LIN {X 0,Y 221.494,Z 504.483,A -85,B 0,C 180,E1 -25357.99,E2 -25357.99} C_VEL
LIN {X 0,Y 227.921,Z 439.207,A -85,B 0,C 180,E1 -25359.51,E2 -25359.51} C_VEL
LIN {X 0,Y 226.419,Z 435.193,A -85,B 0,C 180,E1 -25360.912,E2 -25360.912} C_VEL
LIN {X 0,Y 223.343,Z 428.758,A -85,B 0,C 180,E1 -25364.018,E2 -25364.018} C_VEL
LIN {X 0,Y 220.682,Z 423.431,A -85,B 0,C 180,E1 -25367.335,E2 -25367.335} C_VEL
LIN {X 0,Y 218.87,Z 419.91,A -85,B 0,C 180,E1 -25370.237,E2 -25370.237} C_VEL
LIN {X 0,Y 217.27,Z 416.47,A -85,B 0,C 180,E1 -25373.966,E2 -25373.966} C_VEL
LIN {X 0,Y 216.23,Z 414.392,A -85,B 0,C 180,E1 -25380,E2 -25380} C_VEL
LIN {X 0,Y 217.433,Z 416.799,A -85,B 0,C 180,E1 -25386.962,E2 -25386.962} C_VEL
LIN {X 0,Y 219.423,Z 421.023,A -85,B 0,C 180,E1 -25391.197,E2 -25391.197} C_VEL
LIN {X 0,Y 221.498,Z 425.12,A -85,B 0,C 180,E1 -25394.235,E2 -25394.235} C_VEL
LIN {X 0,Y 223.862,Z 429.779,A -85,B 0,C 180,E1 -25397,E2 -25397} C_VEL
LIN {X 0,Y 227.551,Z 437.653,A -85,B 0,C 180,E1 -25400.561,E2 -25400.561} C_VEL
LIN {X 0,Y 227.966,Z 438.553,A -85,B 0,C 180,E1 -25400.919,E2 -25400.919} C_VEL
LIN {X 0,Y 221.714,Z 501.532,A -85,B 0,C 180,E1 -25402.388,E2 -25402.388} C_VEL
LIN {X 0,Y 218.854,Z 518.054,A -85,B 0,C 180,E1 -25402.945,E2 -25402.945} C_VEL
LIN {X 0,Y 214.898,Z 534.172,A -85,B 0,C 180,E1 -25403.694,E2 -25403.694} C_VEL
LIN {X 0,Y 209.854,Z 550.115,A -85,B 0,C 180,E1 -25404.713,E2 -25404.713} C_VEL
LIN {X 0,Y 204.116,Z 564.778,A -85,B 0,C 180,E1 -25405.906,E2 -25405.906} C_VEL
LIN {X 0,Y 197.233,Z 579.446,A -85,B 0,C 180,E1 -25407.461,E2 -25407.461} C_VEL
LIN {X 0,Y 189.58,Z 593.437,A -85,B 0,C 180,E1 -25409.405,E2 -25409.405} C_VEL
LIN {X 0,Y 181.509,Z 606.104,A -85,B 0,C 180,E1 -25411.589,E2 -25411.589} C_VEL
LIN {X 0,Y 173.842,Z 617.019,A -85,B 0,C 180,E1 -25414.028,E2 -25414.028} C_VEL
LIN {X 0,Y 166.48,Z 626.388,A -85,B 0,C 180,E1 -25416.67,E2 -25416.67} C_VEL
LIN {X 0,Y 157.191,Z 637.123,A -85,B 0,C 180,E1 -25420.53,E2 -25420.53} C_VEL
LIN {X 0,Y 148.617,Z 646.133,A -85,B 0,C 180,E1 -25424.819,E2 -25424.819} C_VEL
LIN {X 0,Y 141.063,Z 653.654,A -85,B 0,C 180,E1 -25429.633,E2 -25429.633} C_VEL
LIN {X 0,Y 132.944,Z 661.201,A -85,B 0,C 180,E1 -25436.284,E2 -25436.284} C_VEL
LIN {X 0,Y 126.667,Z 666.92,A -85,B 0,C 180,E1 -25443.649,E2 -25443.649} C_VEL
LIN {X 0,Y 122.985,Z 670.259,A -85,B 0,C 180,E1 -25449.948,E2 -25449.948} C_VEL
LIN {X 0,Y 120.736,Z 672.675,A -85,B 0,C 180,E1 -25456.536,E2 -25456.536} C_VEL
LIN {X 0,Y 119.59,Z 674.038,A -85,B 0,C 180,E1 -25463.25,E2 -25463.25} C_VEL
LIN {X 0,Y 119.419,Z 674.556,A -85,B 0,C 180,E1 -25470,E2 -25470} C_VEL
LIN {X 0,Y 119.59,Z 674.067,A -85,B 0,C 180,E1 -25476.75,E2 -25476.75} C_VEL
LIN {X 0,Y 120.729,Z 672.734,A -85,B 0,C 180,E1 -25483.465,E2 -25483.465} C_VEL
LIN {X 0,Y 122.952,Z 670.346,A -85,B 0,C 180,E1 -25490.057,E2 -25490.057} C_VEL
LIN {X 0,Y 126.618,Z 667.042,A -85,B 0,C 180,E1 -25496.362,E2 -25496.362} C_VEL
LIN {X 0,Y 132.912,Z 661.357,A -85,B 0,C 180,E1 -25503.725,E2 -25503.725} C_VEL
LIN {X 0,Y 141.009,Z 653.864,A -85,B 0,C 180,E1 -25510.385,E2 -25510.385} C_VEL
LIN {X 0,Y 149.586,Z 645.371,A -85,B 0,C 180,E1 -25515.765,E2 -25515.765} C_VEL
LIN {X 0,Y 158.221,Z 636.189,A -85,B 0,C 180,E1 -25520.015,E2 -25520.015} C_VEL
LIN {X 0,Y 166.39,Z 626.732,A -85,B 0,C 180,E1 -25523.371,E2 -25523.371} C_VEL
LIN {X 0,Y 173.745,Z 617.398,A -85,B 0,C 180,E1 -25526.018,E2 -25526.018} C_VEL
LIN {X 0,Y 181.444,Z 606.553,A -85,B 0,C 180,E1 -25528.445,E2 -25528.445} C_VEL
LIN {X 0,Y 189.51,Z 593.974,A -85,B 0,C 180,E1 -25530.632,E2 -25530.632} C_VEL
LIN {X 0,Y 196.444,Z 581.403,A -85,B 0,C 180,E1 -25532.434,E2 -25532.434} C_VEL
LIN {X 0,Y 203.313,Z 567.081,A -85,B 0,C 180,E1 -25533.993,E2 -25533.993} C_VEL
LIN {X 0,Y 209.066,Z 553.002,A -85,B 0,C 180,E1 -25535.179,E2 -25535.179} C_VEL
LIN {X 0,Y 214.072,Z 537.944,A -85,B 0,C 180,E1 -25536.224,E2 -25536.224} C_VEL
LIN {X 0,Y 218.277,Z 521.791,A -85,B 0,C 180,E1 -25537.037,E2 -25537.037} C_VEL
LIN {X 0,Y 221.319,Z 505.505,A -85,B 0,C 180,E1 -25537.631,E2 -25537.631} C_VEL
LIN {X 0,Y 223.9,Z 483.093,A -85,B 0,C 180,E1 -25538.178,E2 -25538.178} C_VEL
LIN {X 0,Y 228.194,Z 438.76,A -85,B 0,C 180,E1 -25539.19,E2 -25539.19} C_VEL
LIN {X 0,Y 224.904,Z 431.726,A -85,B 0,C 180,E1 -25542.261,E2 -25542.261} C_VEL
LIN {X 0,Y 222.442,Z 426.637,A -85,B 0,C 180,E1 -25545.008,E2 -25545.008} C_VEL
LIN {X 0,Y 220.387,Z 422.756,A -85,B 0,C 180,E1 -25547.766,E2 -25547.766} C_VEL
LIN {X 0,Y 219.16,Z 420.172,A -85,B 0,C 180,E1 -25549.841,E2 -25549.841} C_VEL
LIN {X 0,Y 217.586,Z 416.739,A -85,B 0,C 180,E1 -25553.509,E2 -25553.509} C_VEL
LIN {X 0,Y 216.511,Z 414.774,A -85,B 0,C 180,E1 -25560,E2 -25560} C_VEL
LIN {X 0,Y 217.626,Z 416.867,A -85,B 0,C 180,E1 -25566.257,E2 -25566.257} C_VEL
LIN {X 0,Y 219.235,Z 420.273,A -85,B 0,C 180,E1 -25569.922,E2 -25569.922} C_VEL
LIN {X 0,Y 221.587,Z 425.06,A -85,B 0,C 180,E1 -25573.556,E2 -25573.556} C_VEL
LIN {X 0,Y 224.194,Z 430.159,A -85,B 0,C 180,E1 -25576.621,E2 -25576.621} C_VEL
LIN {X 0,Y 227.397,Z 437.132,A -85,B 0,C 180,E1 -25579.757,E2 -25579.757} C_VEL
LIN {X 0,Y 228.202,Z 439.552,A -85,B 0,C 180,E1 -25580.519,E2 -25580.519} C_VEL
LIN {X 0,Y 221.379,Z 507.429,A -85,B 0,C 180,E1 -25582.062,E2 -25582.062} C_VEL
LIN {X 0,Y 218.386,Z 523.964,A -85,B 0,C 180,E1 -25582.589,E2 -25582.589} C_VEL
LIN {X 0,Y 214.635,Z 538.749,A -85,B 0,C 180,E1 -25583.219,E2 -25583.219} C_VEL
LIN {X 0,Y 209.754,Z 553.938,A -85,B 0,C 180,E1 -25584.073,E2 -25584.073} C_VEL
LIN {X 0,Y 203.894,Z 568.874,A -85,B 0,C 180,E1 -25585.204,E2 -25585.204} C_VEL
LIN {X 0,Y 196.702,Z 584.097,A -85,B 0,C 180,E1 -25586.719,E2 -25586.719} C_VEL
LIN {X 0,Y 188.97,Z 598.053,A -85,B 0,C 180,E1 -25588.523,E2 -25588.523} C_VEL
LIN {X 0,Y 181.019,Z 610.686,A -85,B 0,C 180,E1 -25590.642,E2 -25590.642} C_VEL
LIN {X 0,Y 172.227,Z 622.919,A -85,B 0,C 180,E1 -25593.225,E2 -25593.225} C_VEL
LIN {X 0,Y 170.959,Z 624.557,A -85,B 0,C 180,E1 -25593.648,E2 -25593.648} C_VEL
LIN {X 0,Y 167.411,Z 628.624,A -85,B 0,C 180,E1 -25594.531,E2 -25594.531} C_VEL
LIN {X 0,Y 154.654,Z 639.69,A -85,B 0,C 180,E1 -25596.604,E2 -25596.604} C_VEL
LIN {X 0,Y 150.879,Z 643.086,A -85,B 0,C 180,E1 -25597.69,E2 -25597.69} C_VEL
LIN {X 0,Y 149.826,Z 644.194,A -85,B 0,C 180,E1 -25598.15,E2 -25598.15} C_VEL
LIN {X 0,Y 140.813,Z 653.17,A -85,B 0,C 180,E1 -25602.594,E2 -25602.594} C_VEL
LIN {X 0,Y 132.233,Z 661.232,A -85,B 0,C 180,E1 -25608.079,E2 -25608.079} C_VEL
LIN {X 0,Y 125.287,Z 667.51,A -85,B 0,C 180,E1 -25613.915,E2 -25613.915} C_VEL
LIN {X 0,Y 118.796,Z 673.385,A -85,B 0,C 180,E1 -25621.753,E2 -25621.753} C_VEL
LIN {X 0,Y 115.131,Z 676.828,A -85,B 0,C 180,E1 -25628.515,E2 -25628.515} C_VEL
LIN {X 0,Y 112.881,Z 679.342,A -85,B 0,C 180,E1 -25635.58,E2 -25635.58} C_VEL
LIN {X 0,Y 112.089,Z 680.775,A -85,B 0,C 180,E1 -25642.796,E2 -25642.796} C_VEL
LIN {X 0,Y 112.247,Z 681.32,A -85,B 0,C 180,E1 -25650,E2 -25650} C_VEL
LIN {X 0,Y 112.089,Z 680.758,A -85,B 0,C 180,E1 -25657.204,E2 -25657.204} C_VEL
LIN {X 0,Y 112.88,Z 679.308,A -85,B 0,C 180,E1 -25664.421,E2 -25664.421} C_VEL
LIN {X 0,Y 115.126,Z 676.778,A -85,B 0,C 180,E1 -25671.486,E2 -25671.486} C_VEL
LIN {X 0,Y 118.797,Z 673.315,A -85,B 0,C 180,E1 -25678.247,E2 -25678.247} C_VEL
LIN {X 0,Y 125.305,Z 667.419,A -85,B 0,C 180,E1 -25686.08,E2 -25686.08} C_VEL
LIN {X 0,Y 133.826,Z 659.689,A -85,B 0,C 180,E1 -25693.055,E2 -25693.055} C_VEL
LIN {X 0,Y 142.972,Z 650.99,A -85,B 0,C 180,E1 -25698.558,E2 -25698.558} C_VEL
LIN {X 0,Y 152.135,Z 641.463,A -85,B 0,C 180,E1 -25702.957,E2 -25702.957} C_VEL
LIN {X 0,Y 160.614,Z 631.959,A -85,B 0,C 180,E1 -25706.241,E2 -25706.241} C_VEL
LIN {X 0,Y 169.713,Z 620.726,A -85,B 0,C 180,E1 -25709.235,E2 -25709.235} C_VEL
LIN {X 0,Y 177.632,Z 609.886,A -85,B 0,C 180,E1 -25711.438,E2 -25711.438} C_VEL
LIN {X 0,Y 185.662,Z 597.499,A -85,B 0,C 180,E1 -25713.417,E2 -25713.417} C_VEL
LIN {X 0,Y 193.591,Z 583.464,A -85,B 0,C 180,E1 -25715.173,E2 -25715.173} C_VEL
LIN {X 0,Y 200.242,Z 569.835,A -85,B 0,C 180,E1 -25716.479,E2 -25716.479} C_VEL
LIN {X 0,Y 206.156,Z 555.242,A -85,B 0,C 180,E1 -25717.584,E2 -25717.584} C_VEL
LIN {X 0,Y 211.488,Z 539.146,A -85,B 0,C 180,E1 -25718.508,E2 -25718.508} C_VEL
LIN {X 0,Y 215.729,Z 522.746,A -85,B 0,C 180,E1 -25719.158,E2 -25719.158} C_VEL
LIN {X 0,Y 218.588,Z 507.04,A -85,B 0,C 180,E1 -25719.643,E2 -25719.643} C_VEL
LIN {X 0,Y 225.169,Z 442.849,A -85,B 0,C 180,E1 -25721.097,E2 -25721.097} C_VEL
LIN {X 0,Y 222.528,Z 436.715,A -85,B 0,C 180,E1 -25723.84,E2 -25723.84} C_VEL
LIN {X 0,Y 220.247,Z 431.987,A -85,B 0,C 180,E1 -25726.624,E2 -25726.624} C_VEL
LIN {X 0,Y 217.995,Z 427.146,A -85,B 0,C 180,E1 -25730.197,E2 -25730.197} C_VEL
LIN {X 0,Y 216.24,Z 423.391,A -85,B 0,C 180,E1 -25734.405,E2 -25734.405} C_VEL
LIN {X 0,Y 215.36,Z 421.481,A -85,B 0,C 180,E1 -25740,E2 -25740} C_VEL
LIN {X 0,Y 216.439,Z 423.719,A -85,B 0,C 180,E1 -25746.643,E2 -25746.643} C_VEL
LIN {X 0,Y 218.209,Z 427.737,A -85,B 0,C 180,E1 -25750.677,E2 -25750.677} C_VEL
LIN {X 0,Y 220.094,Z 431.665,A -85,B 0,C 180,E1 -25753.621,E2 -25753.621} C_VEL
LIN {X 0,Y 222.294,Z 436.235,A -85,B 0,C 180,E1 -25756.355,E2 -25756.355} C_VEL
LIN {X 0,Y 225.122,Z 442.608,A -85,B 0,C 180,E1 -25759.3,E2 -25759.3} C_VEL
LIN {X 0,Y 219.149,Z 501.479,A -85,B 0,C 180,E1 -25760.669,E2 -25760.669} C_VEL
LIN {X 0,Y 216.266,Z 517.933,A -85,B 0,C 180,E1 -25761.207,E2 -25761.207} C_VEL
LIN {X 0,Y 212.515,Z 533.145,A -85,B 0,C 180,E1 -25761.883,E2 -25761.883} C_VEL
LIN {X 0,Y 207.706,Z 548.35,A -85,B 0,C 180,E1 -25762.775,E2 -25762.775} C_VEL
LIN {X 0,Y 201.845,Z 563.288,A -85,B 0,C 180,E1 -25763.938,E2 -25763.938} C_VEL
LIN {X 0,Y 195.334,Z 577.121,A -85,B 0,C 180,E1 -25765.314,E2 -25765.314} C_VEL
LIN {X 0,Y 187.563,Z 591.314,A -85,B 0,C 180,E1 -25767.138,E2 -25767.138} C_VEL
LIN {X 0,Y 179.949,Z 603.401,A -85,B 0,C 180,E1 -25769.09,E2 -25769.09} C_VEL
LIN {X 0,Y 171.251,Z 615.5,A -85,B 0,C 180,E1 -25771.619,E2 -25771.619} C_VEL
LIN {X 0,Y 163.137,Z 625.599,A -85,B 0,C 180,E1 -25774.327,E2 -25774.327} C_VEL
LIN {X 0,Y 153.81,Z 636.113,A -85,B 0,C 180,E1 -25777.983,E2 -25777.983} C_VEL
LIN {X 0,Y 144.743,Z 645.342,A -85,B 0,C 180,E1 -25782.23,E2 -25782.23} C_VEL
LIN {X 0,Y 135.692,Z 653.865,A -85,B 0,C 180,E1 -25787.676,E2 -25787.676} C_VEL
LIN {X 0,Y 127.055,Z 661.411,A -85,B 0,C 180,E1 -25794.493,E2 -25794.493} C_VEL
LIN {X 0,Y 120.293,Z 667.13,A -85,B 0,C 180,E1 -25802.135,E2 -25802.135} C_VEL
LIN {X 0,Y 116.294,Z 670.469,A -85,B 0,C 180,E1 -25808.74,E2 -25808.74} C_VEL
LIN {X 0,Y 113.824,Z 672.884,A -85,B 0,C 180,E1 -25815.701,E2 -25815.701} C_VEL
LIN {X 0,Y 112.549,Z 674.245,A -85,B 0,C 180,E1 -25822.826,E2 -25822.826} C_VEL
LIN {X 0,Y 112.335,Z 674.763,A -85,B 0,C 180,E1 -25830,E2 -25830} C_VEL
LIN {X 0,Y 112.549,Z 674.274,A -85,B 0,C 180,E1 -25837.174,E2 -25837.174} C_VEL
LIN {X 0,Y 113.801,Z 672.941,A -85,B 0,C 180,E1 -25844.301,E2 -25844.301} C_VEL
LIN {X 0,Y 116.261,Z 670.555,A -85,B 0,C 180,E1 -25851.266,E2 -25851.266} C_VEL
LIN {X 0,Y 120.246,Z 667.25,A -85,B 0,C 180,E1 -25857.877,E2 -25857.877} C_VEL
LIN {X 0,Y 127.025,Z 661.565,A -85,B 0,C 180,E1 -25865.516,E2 -25865.516} C_VEL
LIN {X 0,Y 135.623,Z 654.072,A -85,B 0,C 180,E1 -25872.35,E2 -25872.35} C_VEL
LIN {X 0,Y 144.681,Z 645.578,A -85,B 0,C 180,E1 -25877.797,E2 -25877.797} C_VEL
LIN {X 0,Y 153.719,Z 636.396,A -85,B 0,C 180,E1 -25882.06,E2 -25882.06} C_VEL
LIN {X 0,Y 162.215,Z 626.939,A -85,B 0,C 180,E1 -25885.404,E2 -25885.404} C_VEL
LIN {X 0,Y 169.857,Z 617.604,A -85,B 0,C 180,E1 -25888.016,E2 -25888.016} C_VEL
LIN {X 0,Y 177.814,Z 606.758,A -85,B 0,C 180,E1 -25890.404,E2 -25890.404} C_VEL
LIN {X 0,Y 186.121,Z 594.178,A -85,B 0,C 180,E1 -25892.544,E2 -25892.544} C_VEL
LIN {X 0,Y 193.159,Z 581.779,A -85,B 0,C 180,E1 -25894.283,E2 -25894.283} C_VEL
LIN {X 0,Y 200.304,Z 567.284,A -85,B 0,C 180,E1 -25895.817,E2 -25895.817} C_VEL
LIN {X 0,Y 206.188,Z 553.203,A -85,B 0,C 180,E1 -25896.969,E2 -25896.969} C_VEL
LIN {X 0,Y 211.316,Z 538.142,A -85,B 0,C 180,E1 -25897.982,E2 -25897.982} C_VEL
LIN {X 0,Y 215.622,Z 521.964,A -85,B 0,C 180,E1 -25898.768,E2 -25898.768} C_VEL
LIN {X 0,Y 218.763,Z 505.415,A -85,B 0,C 180,E1 -25899.358,E2 -25899.358} C_VEL
LIN {X 0,Y 221.455,Z 482.343,A -85,B 0,C 180,E1 -25899.904,E2 -25899.904} C_VEL
LIN {X 0,Y 225.371,Z 442.866,A -85,B 0,C 180,E1 -25900.792,E2 -25900.792} C_VEL
LIN {X 0,Y 222.757,Z 436.94,A -85,B 0,C 180,E1 -25903.504,E2 -25903.504} C_VEL
LIN {X 0,Y 220.658,Z 432.526,A -85,B 0,C 180,E1 -25906.062,E2 -25906.062} C_VEL
LIN {X 0,Y 218.91,Z 428.999,A -85,B 0,C 180,E1 -25908.647,E2 -25908.647} C_VEL
LIN {X 0,Y 217.913,Z 426.828,A -85,B 0,C 180,E1 -25910.486,E2 -25910.486} C_VEL
LIN {X 0,Y 216.559,Z 423.625,A -85,B 0,C 180,E1 -25913.945,E2 -25913.945} C_VEL
LIN {X 0,Y 215.643,Z 421.841,A -85,B 0,C 180,E1 -25920,E2 -25920} C_VEL
LIN {X 0,Y 216.664,Z 423.955,A -85,B 0,C 180,E1 -25926.051,E2 -25926.051} C_VEL
LIN {X 0,Y 218.401,Z 427.814,A -85,B 0,C 180,E1 -25930.077,E2 -25930.077} C_VEL
LIN {X 0,Y 220.496,Z 432.245,A -85,B 0,C 180,E1 -25933.361,E2 -25933.361} C_VEL
LIN {X 0,Y 222.814,Z 437.08,A -85,B 0,C 180,E1 -25936.197,E2 -25936.197} C_VEL
LIN {X 0,Y 225.415,Z 443.085,A -85,B 0,C 180,E1 -25938.895,E2 -25938.895} C_VEL
LIN {X 0,Y 218.88,Z 506.754,A -85,B 0,C 180,E1 -25940.325,E2 -25940.325} C_VEL
LIN {X 0,Y 215.741,Z 523.856,A -85,B 0,C 180,E1 -25940.852,E2 -25940.852} C_VEL
LIN {X 0,Y 211.534,Z 539.938,A -85,B 0,C 180,E1 -25941.525,E2 -25941.525} C_VEL
LIN {X 0,Y 206.201,Z 555.726,A -85,B 0,C 180,E1 -25942.407,E2 -25942.407} C_VEL
LIN {X 0,Y 200.222,Z 570.315,A -85,B 0,C 180,E1 -25943.508,E2 -25943.508} C_VEL
LIN {X 0,Y 192.869,Z 585.319,A -85,B 0,C 180,E1 -25944.985,E2 -25944.985} C_VEL
LIN {X 0,Y 184.949,Z 599.026,A -85,B 0,C 180,E1 -25946.75,E2 -25946.75} C_VEL
LIN {X 0,Y 176.591,Z 611.738,A -85,B 0,C 180,E1 -25948.89,E2 -25948.89} C_VEL
LIN {X 0,Y 167.08,Z 624.349,A -85,B 0,C 180,E1 -25951.594,E2 -25951.594} C_VEL
LIN {X 0,Y 158.129,Z 635.109,A -85,B 0,C 180,E1 -25954.693,E2 -25954.693} C_VEL
LIN {X 0,Y 149.826,Z 644.194,A -85,B 0,C 180,E1 -25958.15,E2 -25958.15} C_VEL
LIN {X 0,Y 146.323,Z 647.5,A -85,B 0,C 180,E1 -25959.465,E2 -25959.465} C_VEL
LIN {X 0,Y 139.117,Z 652.656,A -85,B 0,C 180,E1 -25961.254,E2 -25961.254} C_VEL
LIN {X 0,Y 131.8,Z 657.356,A -85,B 0,C 180,E1 -25963.293,E2 -25963.293} C_VEL
LIN {X 0,Y 128.225,Z 659.95,A -85,B 0,C 180,E1 -25965.027,E2 -25965.027} C_VEL
LIN {X 0,Y 119.533,Z 667.3,A -85,B 0,C 180,E1 -25971.877,E2 -25971.877} C_VEL
LIN {X 0,Y 112.473,Z 673.174,A -85,B 0,C 180,E1 -25980.008,E2 -25980.008} C_VEL
LIN {X 0,Y 108.465,Z 676.619,A -85,B 0,C 180,E1 -25987.122,E2 -25987.122} C_VEL
LIN {X 0,Y 105.943,Z 679.133,A -85,B 0,C 180,E1 -25994.612,E2 -25994.612} C_VEL
LIN {X 0,Y 105.012,Z 680.567,A -85,B 0,C 180,E1 -26002.308,E2 -26002.308} C_VEL
LIN {X 0,Y 105.165,Z 681.114,A -85,B 0,C 180,E1 -26010,E2 -26010} C_VEL
LIN {X 0,Y 105.012,Z 680.55,A -85,B 0,C 180,E1 -26017.692,E2 -26017.692} C_VEL
LIN {X 0,Y 105.941,Z 679.098,A -85,B 0,C 180,E1 -26025.388,E2 -26025.388} C_VEL
LIN {X 0,Y 108.461,Z 676.567,A -85,B 0,C 180,E1 -26032.879,E2 -26032.879} C_VEL
LIN {X 0,Y 112.481,Z 673.104,A -85,B 0,C 180,E1 -26039.99,E2 -26039.99} C_VEL
LIN {X 0,Y 119.552,Z 667.208,A -85,B 0,C 180,E1 -26048.116,E2 -26048.116} C_VEL
LIN {X 0,Y 128.647,Z 659.477,A -85,B 0,C 180,E1 -26055.25,E2 -26055.25} C_VEL
LIN {X 0,Y 138.324,Z 650.778,A -85,B 0,C 180,E1 -26060.789,E2 -26060.789} C_VEL
LIN {X 0,Y 148.282,Z 640.876,A -85,B 0,C 180,E1 -26065.337,E2 -26065.337} C_VEL
LIN {X 0,Y 158.052,Z 630.251,A -85,B 0,C 180,E1 -26068.868,E2 -26068.868} C_VEL
LIN {X 0,Y 166.172,Z 620.515,A -85,B 0,C 180,E1 -26071.352,E2 -26071.352} C_VEL
LIN {X 0,Y 174.87,Z 608.891,A -85,B 0,C 180,E1 -26073.659,E2 -26073.659} C_VEL
LIN {X 0,Y 183.288,Z 596.108,A -85,B 0,C 180,E1 -26075.597,E2 -26075.597} C_VEL
LIN {X 0,Y 191.459,Z 581.821,A -85,B 0,C 180,E1 -26077.26,E2 -26077.26} C_VEL
LIN {X 0,Y 198.281,Z 567.923,A -85,B 0,C 180,E1 -26078.499,E2 -26078.499} C_VEL
LIN {X 0,Y 204.155,Z 553.463,A -85,B 0,C 180,E1 -26079.535,E2 -26079.535} C_VEL
LIN {X 0,Y 209.532,Z 537.119,A -85,B 0,C 180,E1 -26080.403,E2 -26080.403} C_VEL
LIN {X 0,Y 213.707,Z 520.692,A -85,B 0,C 180,E1 -26080.99,E2 -26080.99} C_VEL
LIN {X 0,Y 216.555,Z 504.099,A -85,B 0,C 180,E1 -26081.481,E2 -26081.481} C_VEL
LIN {X 0,Y 222.506,Z 446.86,A -85,B 0,C 180,E1 -26082.757,E2 -26082.757} C_VEL
LIN {X 0,Y 219.934,Z 440.86,A -85,B 0,C 180,E1 -26085.78,E2 -26085.78} C_VEL
LIN {X 0,Y 217.832,Z 436.273,A -85,B 0,C 180,E1 -26088.838,E2 -26088.838} C_VEL
LIN {X 0,Y 216.601,Z 433.528,A -85,B 0,C 180,E1 -26091.134,E2 -26091.134} C_VEL
LIN {X 0,Y 215.375,Z 430.464,A -85,B 0,C 180,E1 -26094.382,E2 -26094.382} C_VEL
LIN {X 0,Y 214.489,Z 428.573,A -85,B 0,C 180,E1 -26100,E2 -26100} C_VEL
LIN {X 0,Y 215.414,Z 430.565,A -85,B 0,C 180,E1 -26106.204,E2 -26106.204} C_VEL
LIN {X 0,Y 217.153,Z 434.775,A -85,B 0,C 180,E1 -26110.42,E2 -26110.42} C_VEL
LIN {X 0,Y 218.792,Z 438.383,A -85,B 0,C 180,E1 -26113.113,E2 -26113.113} C_VEL
LIN {X 0,Y 220.845,Z 442.924,A -85,B 0,C 180,E1 -26115.813,E2 -26115.813} C_VEL
LIN {X 0,Y 222.485,Z 446.827,A -85,B 0,C 180,E1 -26117.678,E2 -26117.678} C_VEL
LIN {X 0,Y 216.748,Z 501.746,A -85,B 0,C 180,E1 -26118.92,E2 -26118.92} C_VEL
LIN {X 0,Y 213.865,Z 517.845,A -85,B 0,C 180,E1 -26119.423,E2 -26119.423} C_VEL
LIN {X 0,Y 209.968,Z 533.394,A -85,B 0,C 180,E1 -26120.09,E2 -26120.09} C_VEL
LIN {X 0,Y 205.061,Z 548.564,A -85,B 0,C 180,E1 -26120.945,E2 -26120.945} C_VEL
LIN {X 0,Y 199.072,Z 563.501,A -85,B 0,C 180,E1 -26122.071,E2 -26122.071} C_VEL
LIN {X 0,Y 192.397,Z 577.334,A -85,B 0,C 180,E1 -26123.397,E2 -26123.397} C_VEL
LIN {X 0,Y 184.422,Z 591.526,A -85,B 0,C 180,E1 -26125.168,E2 -26125.168} C_VEL
LIN {X 0,Y 176.597,Z 603.612,A -85,B 0,C 180,E1 -26127.071,E2 -26127.071} C_VEL
LIN {X 0,Y 167.628,Z 615.711,A -85,B 0,C 180,E1 -26129.546,E2 -26129.546} C_VEL
LIN {X 0,Y 159.61,Z 625.33,A -85,B 0,C 180,E1 -26132.04,E2 -26132.04} C_VEL
LIN {X 0,Y 150.74,Z 635.095,A -85,B 0,C 180,E1 -26135.323,E2 -26135.323} C_VEL
LIN {X 0,Y 141.169,Z 644.459,A -85,B 0,C 180,E1 -26139.497,E2 -26139.497} C_VEL
LIN {X 0,Y 132.484,Z 652.288,A -85,B 0,C 180,E1 -26144.263,E2 -26144.263} C_VEL
LIN {X 0,Y 124.735,Z 658.814,A -85,B 0,C 180,E1 -26149.613,E2 -26149.613} C_VEL
LIN {X 0,Y 118.132,Z 664.087,A -85,B 0,C 180,E1 -26155.585,E2 -26155.585} C_VEL
LIN {X 0,Y 114.014,Z 667.34,A -85,B 0,C 180,E1 -26160.454,E2 -26160.454} C_VEL
LIN {X 0,Y 109.667,Z 670.678,A -85,B 0,C 180,E1 -26167.387,E2 -26167.387} C_VEL
LIN {X 0,Y 106.915,Z 673.093,A -85,B 0,C 180,E1 -26174.755,E2 -26174.755} C_VEL
LIN {X 0,Y 105.5,Z 674.453,A -85,B 0,C 180,E1 -26182.343,E2 -26182.343} C_VEL
LIN {X 0,Y 105.237,Z 674.97,A -85,B 0,C 180,E1 -26190,E2 -26190} C_VEL
LIN {X 0,Y 105.499,Z 674.481,A -85,B 0,C 180,E1 -26197.656,E2 -26197.656} C_VEL
LIN {X 0,Y 106.895,Z 673.15,A -85,B 0,C 180,E1 -26205.247,E2 -26205.247} C_VEL
LIN {X 0,Y 109.635,Z 670.763,A -85,B 0,C 180,E1 -26212.62,E2 -26212.62} C_VEL
LIN {X 0,Y 113.969,Z 667.458,A -85,B 0,C 180,E1 -26219.559,E2 -26219.559} C_VEL
LIN {X 0,Y 121.259,Z 661.773,A -85,B 0,C 180,E1 -26227.485,E2 -26227.485} C_VEL
LIN {X 0,Y 130.404,Z 654.28,A -85,B 0,C 180,E1 -26234.476,E2 -26234.476} C_VEL
LIN {X 0,Y 139.97,Z 645.786,A -85,B 0,C 180,E1 -26239.97,E2 -26239.97} C_VEL
LIN {X 0,Y 149.419,Z 636.603,A -85,B 0,C 180,E1 -26244.228,E2 -26244.228} C_VEL
LIN {X 0,Y 158.247,Z 627.146,A -85,B 0,C 180,E1 -26247.545,E2 -26247.545} C_VEL
LIN {X 0,Y 167.542,Z 616.114,A -85,B 0,C 180,E1 -26250.506,E2 -26250.506} C_VEL
LIN {X 0,Y 175.83,Z 605.021,A -85,B 0,C 180,E1 -26252.789,E2 -26252.789} C_VEL
LIN {X 0,Y 183.633,Z 593.216,A -85,B 0,C 180,E1 -26254.711,E2 -26254.711} C_VEL
LIN {X 0,Y 190.831,Z 580.83,A -85,B 0,C 180,E1 -26256.349,E2 -26256.349} C_VEL
LIN {X 0,Y 198.248,Z 565.909,A -85,B 0,C 180,E1 -26257.84,E2 -26257.84} C_VEL
LIN {X 0,Y 204.259,Z 551.424,A -85,B 0,C 180,E1 -26258.953,E2 -26258.953} C_VEL
LIN {X 0,Y 209.527,Z 535.745,A -85,B 0,C 180,E1 -26259.913,E2 -26259.913} C_VEL
LIN {X 0,Y 213.648,Z 520.09,A -85,B 0,C 180,E1 -26260.617,E2 -26260.617} C_VEL
LIN {X 0,Y 216.735,Z 503.437,A -85,B 0,C 180,E1 -26261.172,E2 -26261.172} C_VEL
LIN {X 0,Y 221.477,Z 459.215,A -85,B 0,C 180,E1 -26262.169,E2 -26262.169} C_VEL
LIN {X 0,Y 222.725,Z 446.978,A -85,B 0,C 180,E1 -26262.437,E2 -26262.437} C_VEL
LIN {X 0,Y 219.947,Z 440.496,A -85,B 0,C 180,E1 -26265.751,E2 -26265.751} C_VEL
LIN {X 0,Y 218.02,Z 436.399,A -85,B 0,C 180,E1 -26268.6,E2 -26268.6} C_VEL
LIN {X 0,Y 216.807,Z 433.658,A -85,B 0,C 180,E1 -26270.907,E2 -26270.907} C_VEL
LIN {X 0,Y 215.541,Z 430.546,A -85,B 0,C 180,E1 -26274.386,E2 -26274.386} C_VEL
LIN {X 0,Y 214.776,Z 428.903,A -85,B 0,C 180,E1 -26280,E2 -26280} C_VEL
LIN {X 0,Y 215.676,Z 430.896,A -85,B 0,C 180,E1 -26285.727,E2 -26285.727} C_VEL
LIN {X 0,Y 217.325,Z 434.793,A -85,B 0,C 180,E1 -26289.775,E2 -26289.775} C_VEL
LIN {X 0,Y 219.513,Z 439.612,A -85,B 0,C 180,E1 -26293.304,E2 -26293.304} C_VEL
LIN {X 0,Y 221.933,Z 445.082,A -85,B 0,C 180,E1 -26296.322,E2 -26296.322} C_VEL
LIN {X 0,Y 222.764,Z 447.124,A -85,B 0,C 180,E1 -26297.245,E2 -26297.245} C_VEL
LIN {X 0,Y 216.525,Z 506.54,A -85,B 0,C 180,E1 -26298.567,E2 -26298.567} C_VEL
LIN {X 0,Y 213.335,Z 523.559,A -85,B 0,C 180,E1 -26299.063,E2 -26299.063} C_VEL
LIN {X 0,Y 209.025,Z 539.738,A -85,B 0,C 180,E1 -26299.707,E2 -26299.707} C_VEL
LIN {X 0,Y 203.561,Z 555.617,A -85,B 0,C 180,E1 -26300.563,E2 -26300.563} C_VEL
LIN {X 0,Y 197.487,Z 570.112,A -85,B 0,C 180,E1 -26301.611,E2 -26301.611} C_VEL
LIN {X 0,Y 189.967,Z 585.116,A -85,B 0,C 180,E1 -26303.036,E2 -26303.036} C_VEL
LIN {X 0,Y 181.845,Z 598.821,A -85,B 0,C 180,E1 -26304.739,E2 -26304.739} C_VEL
LIN {X 0,Y 173.239,Z 611.532,A -85,B 0,C 180,E1 -26306.812,E2 -26306.812} C_VEL
LIN {X 0,Y 163.436,Z 624.142,A -85,B 0,C 180,E1 -26309.451,E2 -26309.451} C_VEL
LIN {X 0,Y 154.144,Z 634.901,A -85,B 0,C 180,E1 -26312.491,E2 -26312.491} C_VEL
LIN {X 0,Y 144.65,Z 644.844,A -85,B 0,C 180,E1 -26316.279,E2 -26316.279} C_VEL
LIN {X 0,Y 134.935,Z 653.979,A -85,B 0,C 180,E1 -26320.956,E2 -26320.956} C_VEL
LIN {X 0,Y 128.225,Z 659.95,A -85,B 0,C 180,E1 -26325.027,E2 -26325.027} C_VEL
LIN {X 0,Y 124.771,Z 662.455,A -85,B 0,C 180,E1 -26326.897,E2 -26326.897} C_VEL
LIN {X 0,Y 112.428,Z 668.953,A -85,B 0,C 180,E1 -26332.287,E2 -26332.287} C_VEL
LIN {X 0,Y 109.113,Z 670.83,A -85,B 0,C 180,E1 -26334.625,E2 -26334.625} C_VEL
LIN {X 0,Y 108.273,Z 671.396,A -85,B 0,C 180,E1 -26335.512,E2 -26335.512} C_VEL
LIN {X 0,Y 103.922,Z 674.808,A -85,B 0,C 180,E1 -26341.746,E2 -26341.746} C_VEL
LIN {X 0,Y 100.267,Z 677.781,A -85,B 0,C 180,E1 -26349.485,E2 -26349.485} C_VEL
LIN {X 0,Y 98.31,Z 679.756,A -85,B 0,C 180,E1 -26357.616,E2 -26357.616} C_VEL
LIN {X 0,Y 97.902,Z 680.744,A -85,B 0,C 180,E1 -26365.884,E2 -26365.884} C_VEL
LIN {X 0,Y 98.07,Z 680.906,A -85,B 0,C 180,E1 -26370,E2 -26370} C_VEL
LIN {X 0,Y 97.931,Z 680.341,A -85,B 0,C 180,E1 -26378.252,E2 -26378.252} C_VEL
LIN {X 0,Y 99.039,Z 678.888,A -85,B 0,C 180,E1 -26386.49,E2 -26386.49} C_VEL
LIN {X 0,Y 101.873,Z 676.357,A -85,B 0,C 180,E1 -26394.452,E2 -26394.452} C_VEL
LIN {X 0,Y 106.302,Z 672.892,A -85,B 0,C 180,E1 -26401.932,E2 -26401.932} C_VEL
LIN {X 0,Y 113.974,Z 666.996,A -85,B 0,C 180,E1 -26410.35,E2 -26410.35} C_VEL
LIN {X 0,Y 123.685,Z 659.265,A -85,B 0,C 180,E1 -26417.619,E2 -26417.619} C_VEL
LIN {X 0,Y 133.905,Z 650.567,A -85,B 0,C 180,E1 -26423.167,E2 -26423.167} C_VEL
LIN {X 0,Y 143.683,Z 641.264,A -85,B 0,C 180,E1 -26427.45,E2 -26427.45} C_VEL
LIN {X 0,Y 153.101,Z 631.535,A -85,B 0,C 180,E1 -26430.713,E2 -26430.713} C_VEL
LIN {X 0,Y 162.871,Z 620.304,A -85,B 0,C 180,E1 -26433.556,E2 -26433.556} C_VEL
LIN {X 0,Y 172.641,Z 607.57,A -85,B 0,C 180,E1 -26435.979,E2 -26435.979} C_VEL
LIN {X 0,Y 181.961,Z 593.54,A -85,B 0,C 180,E1 -26437.966,E2 -26437.966} C_VEL
LIN {X 0,Y 190.348,Z 578.746,A -85,B 0,C 180,E1 -26439.535,E2 -26439.535} C_VEL
LIN {X 0,Y 197.311,Z 564.167,A -85,B 0,C 180,E1 -26440.716,E2 -26440.716} C_VEL
LIN {X 0,Y 203.604,Z 548.173,A -85,B 0,C 180,E1 -26441.714,E2 -26441.714} C_VEL
LIN {X 0,Y 208.506,Z 532.663,A -85,B 0,C 180,E1 -26442.412,E2 -26442.412} C_VEL
LIN {X 0,Y 212.486,Z 515.86,A -85,B 0,C 180,E1 -26442.954,E2 -26442.954} C_VEL
LIN {X 0,Y 215.119,Z 498.264,A -85,B 0,C 180,E1 -26443.404,E2 -26443.404} C_VEL
LIN {X 0,Y 220.043,Z 451.149,A -85,B 0,C 180,E1 -26444.415,E2 -26444.415} C_VEL
LIN {X 0,Y 217.815,Z 445.762,A -85,B 0,C 180,E1 -26447.398,E2 -26447.398} C_VEL
LIN {X 0,Y 215.936,Z 441.365,A -85,B 0,C 180,E1 -26450.635,E2 -26450.635} C_VEL
LIN {X 0,Y 214.357,Z 437.386,A -85,B 0,C 180,E1 -26454.827,E2 -26454.827} C_VEL
LIN {X 0,Y 213.62,Z 435.652,A -85,B 0,C 180,E1 -26460,E2 -26460} C_VEL
LIN {X 0,Y 214.428,Z 437.543,A -85,B 0,C 180,E1 -26465.879,E2 -26465.879} C_VEL
LIN {X 0,Y 215.998,Z 441.585,A -85,B 0,C 180,E1 -26469.96,E2 -26469.96} C_VEL
LIN {X 0,Y 217.584,Z 445.253,A -85,B 0,C 180,E1 -26472.712,E2 -26472.712} C_VEL
LIN {X 0,Y 219.464,Z 449.769,A -85,B 0,C 180,E1 -26475.33,E2 -26475.33} C_VEL
LIN {X 0,Y 220.013,Z 451.106,A -85,B 0,C 180,E1 -26476.009,E2 -26476.009} C_VEL
LIN {X 0,Y 214.448,Z 502.776,A -85,B 0,C 180,E1 -26477.148,E2 -26477.148} C_VEL
LIN {X 0,Y 211.304,Z 519.519,A -85,B 0,C 180,E1 -26477.661,E2 -26477.661} C_VEL
LIN {X 0,Y 207.268,Z 534.818,A -85,B 0,C 180,E1 -26478.303,E2 -26478.303} C_VEL
LIN {X 0,Y 201.879,Z 550.755,A -85,B 0,C 180,E1 -26479.214,E2 -26479.214} C_VEL
LIN {X 0,Y 195.751,Z 565.415,A -85,B 0,C 180,E1 -26480.29,E2 -26480.29} C_VEL
LIN {X 0,Y 188.317,Z 580.148,A -85,B 0,C 180,E1 -26481.703,E2 -26481.703} C_VEL
LIN {X 0,Y 180.045,Z 594.073,A -85,B 0,C 180,E1 -26483.464,E2 -26483.464} C_VEL
LIN {X 0,Y 171.285,Z 606.737,A -85,B 0,C 180,E1 -26485.488,E2 -26485.488} C_VEL
LIN {X 0,Y 162.829,Z 617.652,A -85,B 0,C 180,E1 -26487.772,E2 -26487.772} C_VEL
LIN {X 0,Y 154.604,Z 627.023,A -85,B 0,C 180,E1 -26490.266,E2 -26490.266} C_VEL
LIN {X 0,Y 144.171,Z 637.756,A -85,B 0,C 180,E1 -26494.034,E2 -26494.034} C_VEL
LIN {X 0,Y 134.356,Z 646.765,A -85,B 0,C 180,E1 -26498.314,E2 -26498.314} C_VEL
LIN {X 0,Y 125.453,Z 654.287,A -85,B 0,C 180,E1 -26503.258,E2 -26503.258} C_VEL
LIN {X 0,Y 115.69,Z 661.832,A -85,B 0,C 180,E1 -26510.368,E2 -26510.368} C_VEL
LIN {X 0,Y 107.852,Z 667.549,A -85,B 0,C 180,E1 -26518.58,E2 -26518.58} C_VEL
LIN {X 0,Y 103.116,Z 670.887,A -85,B 0,C 180,E1 -26525.862,E2 -26525.862} C_VEL
LIN {X 0,Y 100.05,Z 673.302,A -85,B 0,C 180,E1 -26533.681,E2 -26533.681} C_VEL
LIN {X 0,Y 98.457,Z 674.661,A -85,B 0,C 180,E1 -26541.792,E2 -26541.792} C_VEL
LIN {X 0,Y 98.15,Z 675.177,A -85,B 0,C 180,E1 -26550,E2 -26550} C_VEL
LIN {X 0,Y 98.456,Z 674.689,A -85,B 0,C 180,E1 -26558.208,E2 -26558.208} C_VEL
LIN {X 0,Y 100.032,Z 673.358,A -85,B 0,C 180,E1 -26566.321,E2 -26566.321} C_VEL
LIN {X 0,Y 103.085,Z 670.97,A -85,B 0,C 180,E1 -26574.146,E2 -26574.146} C_VEL
LIN {X 0,Y 107.807,Z 667.666,A -85,B 0,C 180,E1 -26581.434,E2 -26581.434} C_VEL
LIN {X 0,Y 115.663,Z 661.981,A -85,B 0,C 180,E1 -26589.643,E2 -26589.643} C_VEL
LIN {X 0,Y 125.388,Z 654.488,A -85,B 0,C 180,E1 -26596.773,E2 -26596.773} C_VEL
LIN {X 0,Y 134.295,Z 646.991,A -85,B 0,C 180,E1 -26601.719,E2 -26601.719} C_VEL
LIN {X 0,Y 144.084,Z 638.031,A -85,B 0,C 180,E1 -26606.017,E2 -26606.017} C_VEL
LIN {X 0,Y 154.53,Z 627.353,A -85,B 0,C 180,E1 -26609.781,E2 -26609.781} C_VEL
LIN {X 0,Y 164.147,Z 616.319,A -85,B 0,C 180,E1 -26612.674,E2 -26612.674} C_VEL
LIN {X 0,Y 172.696,Z 605.226,A -85,B 0,C 180,E1 -26614.887,E2 -26614.887} C_VEL
LIN {X 0,Y 180.699,Z 593.421,A -85,B 0,C 180,E1 -26616.758,E2 -26616.758} C_VEL
LIN {X 0,Y 188.041,Z 581.12,A -85,B 0,C 180,E1 -26618.325,E2 -26618.325} C_VEL
LIN {X 0,Y 195.685,Z 566.111,A -85,B 0,C 180,E1 -26619.763,E2 -26619.763} C_VEL
LIN {X 0,Y 201.818,Z 551.625,A -85,B 0,C 180,E1 -26620.835,E2 -26620.835} C_VEL
LIN {X 0,Y 207.197,Z 535.943,A -85,B 0,C 180,E1 -26621.756,E2 -26621.756} C_VEL
LIN {X 0,Y 211.367,Z 520.451,A -85,B 0,C 180,E1 -26622.423,E2 -26622.423} C_VEL
LIN {X 0,Y 214.609,Z 503.331,A -85,B 0,C 180,E1 -26622.967,E2 -26622.967} C_VEL
LIN {X 0,Y 220.268,Z 451.303,A -85,B 0,C 180,E1 -26624.092,E2 -26624.092} C_VEL
LIN {X 0,Y 218.129,Z 446.088,A -85,B 0,C 180,E1 -26626.965,E2 -26626.965} C_VEL
LIN {X 0,Y 215.933,Z 440.871,A -85,B 0,C 180,E1 -26630.87,E2 -26630.87} C_VEL
LIN {X 0,Y 214.535,Z 437.47,A -85,B 0,C 180,E1 -26634.831,E2 -26634.831} C_VEL
LIN {X 0,Y 213.908,Z 435.972,A -85,B 0,C 180,E1 -26640,E2 -26640} C_VEL
LIN {X 0,Y 214.696,Z 437.842,A -85,B 0,C 180,E1 -26645.4,E2 -26645.4} C_VEL
LIN {X 0,Y 216.141,Z 441.517,A -85,B 0,C 180,E1 -26649.238,E2 -26649.238} C_VEL
LIN {X 0,Y 217.826,Z 445.478,A -85,B 0,C 180,E1 -26652.224,E2 -26652.224} C_VEL
LIN {X 0,Y 219.867,Z 450.363,A -85,B 0,C 180,E1 -26655.053,E2 -26655.053} C_VEL
LIN {X 0,Y 220.292,Z 451.358,A -85,B 0,C 180,E1 -26655.57,E2 -26655.57} C_VEL
LIN {X 0,Y 214.305,Z 506.748,A -85,B 0,C 180,E1 -26656.773,E2 -26656.773} C_VEL
LIN {X 0,Y 210.904,Z 524.382,A -85,B 0,C 180,E1 -26657.274,E2 -26657.274} C_VEL
LIN {X 0,Y 206.414,Z 540.607,A -85,B 0,C 180,E1 -26657.901,E2 -26657.901} C_VEL
LIN {X 0,Y 201.127,Z 555.527,A -85,B 0,C 180,E1 -26658.671,E2 -26658.671} C_VEL
LIN {X 0,Y 194.973,Z 569.909,A -85,B 0,C 180,E1 -26659.663,E2 -26659.663} C_VEL
LIN {X 0,Y 187.295,Z 584.912,A -85,B 0,C 180,E1 -26661.03,E2 -26661.03} C_VEL
LIN {X 0,Y 178.974,Z 598.616,A -85,B 0,C 180,E1 -26662.662,E2 -26662.662} C_VEL
LIN {X 0,Y 170.89,Z 610.308,A -85,B 0,C 180,E1 -26664.481,E2 -26664.481} C_VEL
LIN {X 0,Y 161.458,Z 622.299,A -85,B 0,C 180,E1 -26666.833,E2 -26666.833} C_VEL
LIN {X 0,Y 151.769,Z 633.256,A -85,B 0,C 180,E1 -26669.744,E2 -26669.744} C_VEL
LIN {X 0,Y 142.525,Z 642.608,A -85,B 0,C 180,E1 -26673.042,E2 -26673.042} C_VEL
LIN {X 0,Y 133.892,Z 650.719,A -85,B 0,C 180,E1 -26676.826,E2 -26676.826} C_VEL
LIN {X 0,Y 123.667,Z 659.396,A -85,B 0,C 180,E1 -26682.372,E2 -26682.372} C_VEL
LIN {X 0,Y 113.954,Z 667.091,A -85,B 0,C 180,E1 -26689.641,E2 -26689.641} C_VEL
LIN {X 0,Y 108.273,Z 671.396,A -85,B 0,C 180,E1 -26695.512,E2 -26695.512} C_VEL
LIN {X 0,Y 105.508,Z 673.109,A -85,B 0,C 180,E1 -26698.169,E2 -26698.169} C_VEL
LIN {X 0,Y 99.744,Z 675.475,A -85,B 0,C 180,E1 -26702.482,E2 -26702.482} C_VEL
LIN {X 0,Y 95.371,Z 677.04,A -85,B 0,C 180,E1 -26706.286,E2 -26706.286} C_VEL
LIN {X 0,Y 93.066,Z 678.006,A -85,B 0,C 180,E1 -26709.553,E2 -26709.553} C_VEL
LIN {X 0,Y 92.608,Z 678.314,A -85,B 0,C 180,E1 -26710.723,E2 -26710.723} C_VEL
LIN {X 0,Y 90.855,Z 680.15,A -85,B 0,C 180,E1 -26721.1,E2 -26721.1} C_VEL
LIN {X 0,Y 90.968,Z 680.699,A -85,B 0,C 180,E1 -26730,E2 -26730} C_VEL
LIN {X 0,Y 90.855,Z 680.132,A -85,B 0,C 180,E1 -26738.9,E2 -26738.9} C_VEL
LIN {X 0,Y 92.178,Z 678.678,A -85,B 0,C 180,E1 -26747.757,E2 -26747.757} C_VEL
LIN {X 0,Y 95.377,Z 676.146,A -85,B 0,C 180,E1 -26756.239,E2 -26756.239} C_VEL
LIN {X 0,Y 100.253,Z 672.681,A -85,B 0,C 180,E1 -26764.113,E2 -26764.113} C_VEL
LIN {X 0,Y 108.566,Z 666.784,A -85,B 0,C 180,E1 -26772.821,E2 -26772.821} C_VEL
LIN {X 0,Y 118.94,Z 659.053,A -85,B 0,C 180,E1 -26780.188,E2 -26780.188} C_VEL
LIN {X 0,Y 129.72,Z 650.356,A -85,B 0,C 180,E1 -26785.711,E2 -26785.711} C_VEL
LIN {X 0,Y 139.244,Z 641.692,A -85,B 0,C 180,E1 -26789.687,E2 -26789.687} C_VEL
LIN {X 0,Y 149.71,Z 631.323,A -85,B 0,C 180,E1 -26793.117,E2 -26793.117} C_VEL
LIN {X 0,Y 159.82,Z 620.093,A -85,B 0,C 180,E1 -26795.848,E2 -26795.848} C_VEL
LIN {X 0,Y 169.327,Z 608.071,A -85,B 0,C 180,E1 -26798.066,E2 -26798.066} C_VEL
LIN {X 0,Y 178.628,Z 594.505,A -85,B 0,C 180,E1 -26799.941,E2 -26799.941} C_VEL
LIN {X 0,Y 186.404,Z 581.395,A -85,B 0,C 180,E1 -26801.313,E2 -26801.313} C_VEL
LIN {X 0,Y 193.508,Z 567.495,A -85,B 0,C 180,E1 -26802.433,E2 -26802.433} C_VEL
LIN {X 0,Y 199.451,Z 553.474,A -85,B 0,C 180,E1 -26803.337,E2 -26803.337} C_VEL
LIN {X 0,Y 204.639,Z 538.499,A -85,B 0,C 180,E1 -26804.073,E2 -26804.073} C_VEL
LIN {X 0,Y 209.103,Z 522.081,A -85,B 0,C 180,E1 -26804.619,E2 -26804.619} C_VEL
LIN {X 0,Y 212.112,Z 506.37,A -85,B 0,C 180,E1 -26805.054,E2 -26805.054} C_VEL
LIN {X 0,Y 217.744,Z 455.535,A -85,B 0,C 180,E1 -26806.12,E2 -26806.12} C_VEL
LIN {X 0,Y 215.642,Z 450.223,A -85,B 0,C 180,E1 -26809.437,E2 -26809.437} C_VEL
LIN {X 0,Y 214.314,Z 446.984,A -85,B 0,C 180,E1 -26812.226,E2 -26812.226} C_VEL
LIN {X 0,Y 213.354,Z 444.286,A -85,B 0,C 180,E1 -26815.277,E2 -26815.277} C_VEL
LIN {X 0,Y 212.745,Z 442.779,A -85,B 0,C 180,E1 -26820.473,E2 -26820.473} C_VEL
LIN {X 0,Y 213.481,Z 444.602,A -85,B 0,C 180,E1 -26825.668,E2 -26825.668} C_VEL
LIN {X 0,Y 214.864,Z 448.352,A -85,B 0,C 180,E1 -26829.496,E2 -26829.496} C_VEL
LIN {X 0,Y 216.384,Z 452.146,A -85,B 0,C 180,E1 -26832.307,E2 -26832.307} C_VEL
LIN {X 0,Y 217.698,Z 455.45,A -85,B 0,C 180,E1 -26834.276,E2 -26834.276} C_VEL
LIN {X 0,Y 212.693,Z 501.27,A -85,B 0,C 180,E1 -26835.281,E2 -26835.281} C_VEL
LIN {X 0,Y 209.638,Z 517.993,A -85,B 0,C 180,E1 -26835.754,E2 -26835.754} C_VEL
LIN {X 0,Y 205.511,Z 533.901,A -85,B 0,C 180,E1 -26836.384,E2 -26836.384} C_VEL
LIN {X 0,Y 200.427,Z 548.991,A -85,B 0,C 180,E1 -26837.153,E2 -26837.153} C_VEL
LIN {X 0,Y 194.19,Z 563.926,A -85,B 0,C 180,E1 -26838.192,E2 -26838.192} C_VEL
LIN {X 0,Y 187.206,Z 577.758,A -85,B 0,C 180,E1 -26839.4,E2 -26839.4} C_VEL
LIN {X 0,Y 178.822,Z 591.95,A -85,B 0,C 180,E1 -26841.028,E2 -26841.028} C_VEL
LIN {X 0,Y 169.849,Z 605.006,A -85,B 0,C 180,E1 -26842.978,E2 -26842.978} C_VEL
LIN {X 0,Y 161.074,Z 616.133,A -85,B 0,C 180,E1 -26845.128,E2 -26845.128} C_VEL
LIN {X 0,Y 151.116,Z 627.235,A -85,B 0,C 180,E1 -26847.916,E2 -26847.916} C_VEL
LIN {X 0,Y 140.298,Z 637.966,A -85,B 0,C 180,E1 -26851.616,E2 -26851.616} C_VEL
LIN {X 0,Y 130.034,Z 646.976,A -85,B 0,C 180,E1 -26855.835,E2 -26855.835} C_VEL
LIN {X 0,Y 120.65,Z 654.498,A -85,B 0,C 180,E1 -26860.777,E2 -26860.777} C_VEL
LIN {X 0,Y 110.262,Z 662.042,A -85,B 0,C 180,E1 -26867.99,E2 -26867.99} C_VEL
LIN {X 0,Y 101.819,Z 667.759,A -85,B 0,C 180,E1 -26876.482,E2 -26876.482} C_VEL
LIN {X 0,Y 96.65,Z 671.096,A -85,B 0,C 180,E1 -26884.132,E2 -26884.132} C_VEL
LIN {X 0,Y 93.232,Z 673.51,A -85,B 0,C 180,E1 -26892.451,E2 -26892.451} C_VEL
LIN {X 0,Y 91.411,Z 674.869,A -85,B 0,C 180,E1 -26901.155,E2 -26901.155} C_VEL
LIN {X 0,Y 91.056,Z 675.384,A -85,B 0,C 180,E1 -26910,E2 -26910} C_VEL
LIN {X 0,Y 91.41,Z 674.897,A -85,B 0,C 180,E1 -26918.845,E2 -26918.845} C_VEL
LIN {X 0,Y 93.199,Z 673.566,A -85,B 0,C 180,E1 -26927.555,E2 -26927.555} C_VEL
LIN {X 0,Y 96.62,Z 671.178,A -85,B 0,C 180,E1 -26935.876,E2 -26935.876} C_VEL
LIN {X 0,Y 103.003,Z 667.008,A -85,B 0,C 180,E1 -26945.037,E2 -26945.037} C_VEL
LIN {X 0,Y 110.222,Z 662.19,A -85,B 0,C 180,E1 -26952.028,E2 -26952.028} C_VEL
LIN {X 0,Y 120.591,Z 654.696,A -85,B 0,C 180,E1 -26959.255,E2 -26959.255} C_VEL
LIN {X 0,Y 131.218,Z 646.2,A -85,B 0,C 180,E1 -26964.763,E2 -26964.763} C_VEL
LIN {X 0,Y 141.548,Z 637.016,A -85,B 0,C 180,E1 -26968.923,E2 -26968.923} C_VEL
LIN {X 0,Y 151.051,Z 627.559,A -85,B 0,C 180,E1 -26972.13,E2 -26972.13} C_VEL
LIN {X 0,Y 160.995,Z 616.524,A -85,B 0,C 180,E1 -26974.931,E2 -26974.931} C_VEL
LIN {X 0,Y 169.8,Z 605.43,A -85,B 0,C 180,E1 -26977.061,E2 -26977.061} C_VEL
LIN {X 0,Y 178.01,Z 593.625,A -85,B 0,C 180,E1 -26978.864,E2 -26978.864} C_VEL
LIN {X 0,Y 185.514,Z 581.345,A -85,B 0,C 180,E1 -26980.369,E2 -26980.369} C_VEL
LIN {X 0,Y 193.347,Z 566.313,A -85,B 0,C 180,E1 -26981.734,E2 -26981.734} C_VEL
LIN {X 0,Y 199.594,Z 551.827,A -85,B 0,C 180,E1 -26982.765,E2 -26982.765} C_VEL
LIN {X 0,Y 205.084,Z 536.143,A -85,B 0,C 180,E1 -26983.642,E2 -26983.642} C_VEL
LIN {X 0,Y 209.34,Z 520.598,A -85,B 0,C 180,E1 -26984.28,E2 -26984.28} C_VEL
LIN {X 0,Y 212.621,Z 503.642,A -85,B 0,C 180,E1 -26984.789,E2 -26984.789} C_VEL
LIN {X 0,Y 217.963,Z 455.698,A -85,B 0,C 180,E1 -26985.813,E2 -26985.813} C_VEL
LIN {X 0,Y 216.089,Z 450.948,A -85,B 0,C 180,E1 -26988.747,E2 -26988.747} C_VEL
LIN {X 0,Y 214.535,Z 447.11,A -85,B 0,C 180,E1 -26991.997,E2 -26991.997} C_VEL
LIN {X 0,Y 213.669,Z 444.553,A -85,B 0,C 180,E1 -26994.81,E2 -26994.81} C_VEL
LIN {X 0,Y 213.04,Z 443.044,A -85,B 0,C 180,E1 -27000,E2 -27000} C_VEL
LIN {X 0,Y 213.724,Z 444.77,A -85,B 0,C 180,E1 -27005.07,E2 -27005.07} C_VEL
LIN {X 0,Y 215.016,Z 448.31,A -85,B 0,C 180,E1 -27008.777,E2 -27008.777} C_VEL
LIN {X 0,Y 216.922,Z 453.016,A -85,B 0,C 180,E1 -27012.275,E2 -27012.275} C_VEL
LIN {X 0,Y 218.012,Z 455.831,A -85,B 0,C 180,E1 -27013.89,E2 -27013.89} C_VEL
LIN {X 0,Y 212.364,Z 506.545,A -85,B 0,C 180,E1 -27014.936,E2 -27014.936} C_VEL
LIN {X 0,Y 208.908,Z 524.176,A -85,B 0,C 180,E1 -27015.413,E2 -27015.413} C_VEL
LIN {X 0,Y 204.311,Z 540.517,A -85,B 0,C 180,E1 -27016.011,E2 -27016.011} C_VEL
LIN {X 0,Y 198.914,Z 555.443,A -85,B 0,C 180,E1 -27016.734,E2 -27016.734} C_VEL
LIN {X 0,Y 192.699,Z 569.706,A -85,B 0,C 180,E1 -27017.673,E2 -27017.673} C_VEL
LIN {X 0,Y 184.853,Z 584.708,A -85,B 0,C 180,E1 -27018.964,E2 -27018.964} C_VEL
LIN {X 0,Y 176.333,Z 598.41,A -85,B 0,C 180,E1 -27020.51,E2 -27020.51} C_VEL
LIN {X 0,Y 167.265,Z 611.119,A -85,B 0,C 180,E1 -27022.426,E2 -27022.426} C_VEL
LIN {X 0,Y 156.888,Z 623.728,A -85,B 0,C 180,E1 -27024.89,E2 -27024.89} C_VEL
LIN {X 0,Y 146.926,Z 634.486,A -85,B 0,C 180,E1 -27027.76,E2 -27027.76} C_VEL
LIN {X 0,Y 136.115,Z 644.884,A -85,B 0,C 180,E1 -27031.578,E2 -27031.578} C_VEL
LIN {X 0,Y 125.949,Z 653.561,A -85,B 0,C 180,E1 -27035.992,E2 -27035.992} C_VEL
LIN {X 0,Y 116.483,Z 660.997,A -85,B 0,C 180,E1 -27041.309,E2 -27041.309} C_VEL
LIN {X 0,Y 108.541,Z 666.881,A -85,B 0,C 180,E1 -27047.167,E2 -27047.167} C_VEL
LIN {X 0,Y 100.246,Z 672.755,A -85,B 0,C 180,E1 -27055.885,E2 -27055.885} C_VEL
LIN {X 0,Y 95.383,Z 676.2,A -85,B 0,C 180,E1 -27063.763,E2 -27063.763} C_VEL
LIN {X 0,Y 92.608,Z 678.314,A -85,B 0,C 180,E1 -27070.723,E2 -27070.723} C_VEL
LIN {X 0,Y 91.137,Z 679.157,A -85,B 0,C 180,E1 -27074.249,E2 -27074.249} C_VEL
LIN {X 0,Y 87.757,Z 680.116,A -85,B 0,C 180,E1 -27080.17,E2 -27080.17} C_VEL
LIN {X 0,Y 84.306,Z 680.522,A -85,B 0,C 180,E1 -27087.828,E2 -27087.828} C_VEL
LIN {X 0,Y 83.824,Z 680.473,A -85,B 0,C 180,E1 -27090.531,E2 -27090.531} C_VEL
LIN {X 0,Y 83.806,Z 679.923,A -85,B 0,C 180,E1 -27099.655,E2 -27099.655} C_VEL
LIN {X 0,Y 85.368,Z 678.468,A -85,B 0,C 180,E1 -27109.227,E2 -27109.227} C_VEL
LIN {X 0,Y 88.988,Z 675.936,A -85,B 0,C 180,E1 -27118.285,E2 -27118.285} C_VEL
LIN {X 0,Y 94.368,Z 672.469,A -85,B 0,C 180,E1 -27126.569,E2 -27126.569} C_VEL
LIN {X 0,Y 103.388,Z 666.572,A -85,B 0,C 180,E1 -27135.541,E2 -27135.541} C_VEL
LIN {X 0,Y 114.461,Z 658.841,A -85,B 0,C 180,E1 -27142.959,E2 -27142.959} C_VEL
LIN {X 0,Y 125.791,Z 650.143,A -85,B 0,C 180,E1 -27148.432,E2 -27148.432} C_VEL
LIN {X 0,Y 136.585,Z 640.757,A -85,B 0,C 180,E1 -27152.572,E2 -27152.572} C_VEL
LIN {X 0,Y 146.61,Z 631.111,A -85,B 0,C 180,E1 -27155.615,E2 -27155.615} C_VEL
LIN {X 0,Y 157.027,Z 619.881,A -85,B 0,C 180,E1 -27158.232,E2 -27158.232} C_VEL
LIN {X 0,Y 166.91,Z 607.709,A -85,B 0,C 180,E1 -27160.365,E2 -27160.365} C_VEL
LIN {X 0,Y 176.314,Z 594.294,A -85,B 0,C 180,E1 -27162.113,E2 -27162.113} C_VEL
LIN {X 0,Y 184.244,Z 581.182,A -85,B 0,C 180,E1 -27163.413,E2 -27163.413} C_VEL
LIN {X 0,Y 191.474,Z 567.281,A -85,B 0,C 180,E1 -27164.47,E2 -27164.47} C_VEL
LIN {X 0,Y 198.019,Z 552.067,A -85,B 0,C 180,E1 -27165.375,E2 -27165.375} C_VEL
LIN {X 0,Y 203.224,Z 536.983,A -85,B 0,C 180,E1 -27166.041,E2 -27166.041} C_VEL
LIN {X 0,Y 207.746,Z 520.028,A -85,B 0,C 180,E1 -27166.556,E2 -27166.556} C_VEL
LIN {X 0,Y 210.806,Z 503.059,A -85,B 0,C 180,E1 -27166.988,E2 -27166.988} C_VEL
LIN {X 0,Y 215.612,Z 460.144,A -85,B 0,C 180,E1 -27167.864,E2 -27167.864} C_VEL
LIN {X 0,Y 213.917,Z 455.654,A -85,B 0,C 180,E1 -27171.022,E2 -27171.022} C_VEL
LIN {X 0,Y 213.155,Z 453.616,A -85,B 0,C 180,E1 -27172.898,E2 -27172.898} C_VEL
LIN {X 0,Y 212.365,Z 451.187,A -85,B 0,C 180,E1 -27175.73,E2 -27175.73} C_VEL
LIN {X 0,Y 211.875,Z 449.865,A -85,B 0,C 180,E1 -27180.475,E2 -27180.475} C_VEL
LIN {X 0,Y 212.512,Z 451.542,A -85,B 0,C 180,E1 -27185.337,E2 -27185.337} C_VEL
LIN {X 0,Y 213.719,Z 455.129,A -85,B 0,C 180,E1 -27188.987,E2 -27188.987} C_VEL
LIN {X 0,Y 215.205,Z 459.033,A -85,B 0,C 180,E1 -27191.909,E2 -27191.909} C_VEL
LIN {X 0,Y 215.6,Z 460.129,A -85,B 0,C 180,E1 -27192.576,E2 -27192.576} C_VEL
LIN {X 0,Y 210.73,Z 503.058,A -85,B 0,C 180,E1 -27193.46,E2 -27193.46} C_VEL
LIN {X 0,Y 207.465,Z 519.868,A -85,B 0,C 180,E1 -27193.928,E2 -27193.928} C_VEL
LIN {X 0,Y 203.266,Z 535.248,A -85,B 0,C 180,E1 -27194.51,E2 -27194.51} C_VEL
LIN {X 0,Y 197.658,Z 551.183,A -85,B 0,C 180,E1 -27195.321,E2 -27195.321} C_VEL
LIN {X 0,Y 191.295,Z 565.84,A -85,B 0,C 180,E1 -27196.301,E2 -27196.301} C_VEL
LIN {X 0,Y 183.437,Z 580.741,A -85,B 0,C 180,E1 -27197.585,E2 -27197.585} C_VEL
LIN {X 0,Y 174.86,Z 594.496,A -85,B 0,C 180,E1 -27199.177,E2 -27199.177} C_VEL
LIN {X 0,Y 165.661,Z 607.159,A -85,B 0,C 180,E1 -27201.041,E2 -27201.041} C_VEL
LIN {X 0,Y 156.698,Z 618.074,A -85,B 0,C 180,E1 -27203.157,E2 -27203.157} C_VEL
LIN {X 0,Y 146.494,Z 628.919,A -85,B 0,C 180,E1 -27205.905,E2 -27205.905} C_VEL
LIN {X 0,Y 136.683,Z 638.177,A -85,B 0,C 180,E1 -27209.061,E2 -27209.061} C_VEL
LIN {X 0,Y 125.981,Z 647.186,A -85,B 0,C 180,E1 -27213.197,E2 -27213.197} C_VEL
LIN {X 0,Y 116.097,Z 654.708,A -85,B 0,C 180,E1 -27218.098,E2 -27218.098} C_VEL
LIN {X 0,Y 105.035,Z 662.253,A -85,B 0,C 180,E1 -27225.367,E2 -27225.367} C_VEL
LIN {X 0,Y 95.921,Z 667.969,A -85,B 0,C 180,E1 -27234.116,E2 -27234.116} C_VEL
LIN {X 0,Y 90.286,Z 671.304,A -85,B 0,C 180,E1 -27242.157,E2 -27242.157} C_VEL
LIN {X 0,Y 86.434,Z 673.719,A -85,B 0,C 180,E1 -27251.02,E2 -27251.02} C_VEL
LIN {X 0,Y 84.394,Z 675.077,A -85,B 0,C 180,E1 -27260.412,E2 -27260.412} C_VEL
LIN {X 0,Y 83.955,Z 675.591,A -85,B 0,C 180,E1 -27270,E2 -27270} C_VEL
LIN {X 0,Y 84.393,Z 675.104,A -85,B 0,C 180,E1 -27279.587,E2 -27279.587} C_VEL
LIN {X 0,Y 86.403,Z 673.774,A -85,B 0,C 180,E1 -27288.987,E2 -27288.987} C_VEL
LIN {X 0,Y 90.242,Z 671.386,A -85,B 0,C 180,E1 -27297.857,E2 -27297.857} C_VEL
LIN {X 0,Y 96.879,Z 667.439,A -85,B 0,C 180,E1 -27307.061,E2 -27307.061} C_VEL
LIN {X 0,Y 104.996,Z 662.399,A -85,B 0,C 180,E1 -27314.654,E2 -27314.654} C_VEL
LIN {X 0,Y 116.04,Z 654.904,A -85,B 0,C 180,E1 -27321.937,E2 -27321.937} C_VEL
LIN {X 0,Y 127.225,Z 646.408,A -85,B 0,C 180,E1 -27327.396,E2 -27327.396} C_VEL
LIN {X 0,Y 137.996,Z 637.222,A -85,B 0,C 180,E1 -27331.464,E2 -27331.464} C_VEL
LIN {X 0,Y 148.685,Z 626.903,A -85,B 0,C 180,E1 -27334.823,E2 -27334.823} C_VEL
LIN {X 0,Y 159.588,Z 614.959,A -85,B 0,C 180,E1 -27337.638,E2 -27337.638} C_VEL
LIN {X 0,Y 169.442,Z 602.6,A -85,B 0,C 180,E1 -27339.787,E2 -27339.787} C_VEL
LIN {X 0,Y 178.774,Z 588.922,A -85,B 0,C 180,E1 -27341.669,E2 -27341.669} C_VEL
LIN {X 0,Y 187.274,Z 574.314,A -85,B 0,C 180,E1 -27343.127,E2 -27343.127} C_VEL
LIN {X 0,Y 194.426,Z 559.612,A -85,B 0,C 180,E1 -27344.242,E2 -27344.242} C_VEL
LIN {X 0,Y 200.403,Z 544.652,A -85,B 0,C 180,E1 -27345.148,E2 -27345.148} C_VEL
LIN {X 0,Y 205.414,Z 528.899,A -85,B 0,C 180,E1 -27345.886,E2 -27345.886} C_VEL
LIN {X 0,Y 209.353,Z 512.485,A -85,B 0,C 180,E1 -27346.419,E2 -27346.419} C_VEL
LIN {X 0,Y 211.987,Z 495.446,A -85,B 0,C 180,E1 -27346.846,E2 -27346.846} C_VEL
LIN {X 0,Y 215.833,Z 460.235,A -85,B 0,C 180,E1 -27347.579,E2 -27347.579} C_VEL
LIN {X 0,Y 214.282,Z 456.226,A -85,B 0,C 180,E1 -27350.442,E2 -27350.442} C_VEL
LIN {X 0,Y 213.47,Z 453.948,A -85,B 0,C 180,E1 -27352.432,E2 -27352.432} C_VEL
LIN {X 0,Y 212.68,Z 451.441,A -85,B 0,C 180,E1 -27355.261,E2 -27355.261} C_VEL
LIN {X 0,Y 212.171,Z 450.118,A -85,B 0,C 180,E1 -27360,E2 -27360} C_VEL
LIN {X 0,Y 212.755,Z 451.737,A -85,B 0,C 180,E1 -27364.737,E2 -27364.737} C_VEL
LIN {X 0,Y 213.931,Z 455.206,A -85,B 0,C 180,E1 -27368.382,E2 -27368.382} C_VEL
LIN {X 0,Y 215.638,Z 459.698,A -85,B 0,C 180,E1 -27371.73,E2 -27371.73} C_VEL
LIN {X 0,Y 215.868,Z 460.339,A -85,B 0,C 180,E1 -27372.114,E2 -27372.114} C_VEL
LIN {X 0,Y 210.671,Z 506.188,A -85,B 0,C 180,E1 -27373.064,E2 -27373.064} C_VEL
LIN {X 0,Y 207.131,Z 523.98,A -85,B 0,C 180,E1 -27373.516,E2 -27373.516} C_VEL
LIN {X 0,Y 202.598,Z 539.874,A -85,B 0,C 180,E1 -27374.053,E2 -27374.053} C_VEL
LIN {X 0,Y 196.935,Z 555.37,A -85,B 0,C 180,E1 -27374.763,E2 -27374.763} C_VEL
LIN {X 0,Y 189.846,Z 571.088,A -85,B 0,C 180,E1 -27375.741,E2 -27375.741} C_VEL
LIN {X 0,Y 181.866,Z 585.821,A -85,B 0,C 180,E1 -27376.977,E2 -27376.977} C_VEL
LIN {X 0,Y 173.183,Z 599.384,A -85,B 0,C 180,E1 -27378.453,E2 -27378.453} C_VEL
LIN {X 0,Y 164.661,Z 610.913,A -85,B 0,C 180,E1 -27380.118,E2 -27380.118} C_VEL
LIN {X 0,Y 155.524,Z 621.887,A -85,B 0,C 180,E1 -27382.124,E2 -27382.124} C_VEL
LIN {X 0,Y 145.172,Z 632.841,A -85,B 0,C 180,E1 -27384.81,E2 -27384.81} C_VEL
LIN {X 0,Y 134.261,Z 643.038,A -85,B 0,C 180,E1 -27388.244,E2 -27388.244} C_VEL
LIN {X 0,Y 124.464,Z 651.318,A -85,B 0,C 180,E1 -27392.115,E2 -27392.115} C_VEL
LIN {X 0,Y 114.434,Z 658.977,A -85,B 0,C 180,E1 -27397.023,E2 -27397.023} C_VEL
LIN {X 0,Y 103.361,Z 666.671,A -85,B 0,C 180,E1 -27404.444,E2 -27404.444} C_VEL
LIN {X 0,Y 94.363,Z 672.545,A -85,B 0,C 180,E1 -27413.429,E2 -27413.429} C_VEL
LIN {X 0,Y 88.993,Z 675.991,A -85,B 0,C 180,E1 -27421.717,E2 -27421.717} C_VEL
LIN {X 0,Y 85.37,Z 678.505,A -85,B 0,C 180,E1 -27430.774,E2 -27430.774} C_VEL
LIN {X 0,Y 83.806,Z 679.942,A -85,B 0,C 180,E1 -27440.345,E2 -27440.345} C_VEL
LIN {X 0,Y 83.873,Z 680.492,A -85,B 0,C 180,E1 -27450,E2 -27450} C_VEL
LIN {X 0,Y 83.824,Z 680.473,A -85,B 0,C 180,E1 -27450.531,E2 -27450.531} C_VEL
LIN {X 0,Y 82.941,Z 680.329,A -85,B 0,C 180,E1 -27454.539,E2 -27454.539} C_VEL
LIN {X 0,Y 80.315,Z 679.715,A -85,B 0,C 180,E1 -27461.25,E2 -27461.25} C_VEL
LIN {X 0,Y 78.73,Z 678.968,A -85,B 0,C 180,E1 -27466.882,E2 -27466.882} C_VEL
LIN {X 0,Y 78.779,Z 678.207,A -85,B 0,C 180,E1 -27471.181,E2 -27471.181} C_VEL
LIN {X 0,Y 79.149,Z 677.886,A -85,B 0,C 180,E1 -27472.58,E2 -27472.58} C_VEL
LIN {X 0,Y 84.59,Z 674.66,A -85,B 0,C 180,E1 -27483.818,E2 -27483.818} C_VEL
LIN {X 0,Y 92.305,Z 670.088,A -85,B 0,C 180,E1 -27493.255,E2 -27493.255} C_VEL
LIN {X 0,Y 100.681,Z 664.919,A -85,B 0,C 180,E1 -27500.161,E2 -27500.161} C_VEL
LIN {X 0,Y 110.273,Z 658.63,A -85,B 0,C 180,E1 -27505.947,E2 -27505.947} C_VEL
LIN {X 0,Y 122.172,Z 649.931,A -85,B 0,C 180,E1 -27511.313,E2 -27511.313} C_VEL
LIN {X 0,Y 131.973,Z 641.786,A -85,B 0,C 180,E1 -27514.864,E2 -27514.864} C_VEL
LIN {X 0,Y 143.792,Z 630.899,A -85,B 0,C 180,E1 -27518.224,E2 -27518.224} C_VEL
LIN {X 0,Y 154.514,Z 619.669,A -85,B 0,C 180,E1 -27520.699,E2 -27520.699} C_VEL
LIN {X 0,Y 165.155,Z 606.828,A -85,B 0,C 180,E1 -27522.81,E2 -27522.81} C_VEL
LIN {X 0,Y 175.057,Z 592.904,A -85,B 0,C 180,E1 -27524.477,E2 -27524.477} C_VEL
LIN {X 0,Y 183.966,Z 578.108,A -85,B 0,C 180,E1 -27525.787,E2 -27525.787} C_VEL
LIN {X 0,Y 191.316,Z 563.526,A -85,B 0,C 180,E1 -27526.774,E2 -27526.774} C_VEL
LIN {X 0,Y 197.867,Z 547.762,A -85,B 0,C 180,E1 -27527.574,E2 -27527.574} C_VEL
LIN {X 0,Y 203.083,Z 532.012,A -85,B 0,C 180,E1 -27528.156,E2 -27528.156} C_VEL
LIN {X 0,Y 207.24,Z 515.2,A -85,B 0,C 180,E1 -27528.6,E2 -27528.6} C_VEL
LIN {X 0,Y 210.017,Z 497.614,A -85,B 0,C 180,E1 -27528.993,E2 -27528.993} C_VEL
LIN {X 0,Y 213.672,Z 464.96,A -85,B 0,C 180,E1 -27529.619,E2 -27529.619} C_VEL
LIN {X 0,Y 212.231,Z 460.737,A -85,B 0,C 180,E1 -27532.986,E2 -27532.986} C_VEL
LIN {X 0,Y 211.469,Z 458.228,A -85,B 0,C 180,E1 -27535.831,E2 -27535.831} C_VEL
LIN {X 0,Y 211.011,Z 456.902,A -85,B 0,C 180,E1 -27540,E2 -27540} C_VEL
LIN {X 0,Y 211.551,Z 458.469,A -85,B 0,C 180,E1 -27545.003,E2 -27545.003} C_VEL
LIN {X 0,Y 212.628,Z 461.974,A -85,B 0,C 180,E1 -27548.554,E2 -27548.554} C_VEL
LIN {X 0,Y 213.654,Z 464.931,A -85,B 0,C 180,E1 -27550.805,E2 -27550.805} C_VEL
LIN {X 0,Y 209.19,Z 503.326,A -85,B 0,C 180,E1 -27551.575,E2 -27551.575} C_VEL
LIN {X 0,Y 205.834,Z 520.276,A -85,B 0,C 180,E1 -27552.022,E2 -27552.022} C_VEL
LIN {X 0,Y 201.609,Z 535.463,A -85,B 0,C 180,E1 -27552.562,E2 -27552.562} C_VEL
LIN {X 0,Y 195.901,Z 551.397,A -85,B 0,C 180,E1 -27553.318,E2 -27553.318} C_VEL
LIN {X 0,Y 189.428,Z 566.052,A -85,B 0,C 180,E1 -27554.243,E2 -27554.243} C_VEL
LIN {X 0,Y 181.301,Z 581.166,A -85,B 0,C 180,E1 -27555.47,E2 -27555.47} C_VEL
LIN {X 0,Y 172.654,Z 594.708,A -85,B 0,C 180,E1 -27556.947,E2 -27556.947} C_VEL
LIN {X 0,Y 163.246,Z 607.369,A -85,B 0,C 180,E1 -27558.714,E2 -27558.714} C_VEL
LIN {X 0,Y 154.025,Z 618.285,A -85,B 0,C 180,E1 -27560.709,E2 -27560.709} C_VEL
LIN {X 0,Y 143.491,Z 629.149,A -85,B 0,C 180,E1 -27563.337,E2 -27563.337} C_VEL
LIN {X 0,Y 133.349,Z 638.388,A -85,B 0,C 180,E1 -27566.368,E2 -27566.368} C_VEL
LIN {X 0,Y 122.21,Z 647.397,A -85,B 0,C 180,E1 -27570.389,E2 -27570.389} C_VEL
LIN {X 0,Y 111.818,Z 654.919,A -85,B 0,C 180,E1 -27575.207,E2 -27575.207} C_VEL
LIN {X 0,Y 100.062,Z 662.464,A -85,B 0,C 180,E1 -27582.483,E2 -27582.483} C_VEL
LIN {X 0,Y 90.212,Z 668.179,A -85,B 0,C 180,E1 -27591.447,E2 -27591.447} C_VEL
LIN {X 0,Y 84.019,Z 671.514,A -85,B 0,C 180,E1 -27599.875,E2 -27599.875} C_VEL
LIN {X 0,Y 79.704,Z 673.929,A -85,B 0,C 180,E1 -27609.347,E2 -27609.347} C_VEL
LIN {X 0,Y 77.386,Z 675.285,A -85,B 0,C 180,E1 -27619.535,E2 -27619.535} C_VEL
LIN {X 0,Y 76.882,Z 675.798,A -85,B 0,C 180,E1 -27630,E2 -27630} C_VEL
LIN {X 0,Y 77.384,Z 675.312,A -85,B 0,C 180,E1 -27640.465,E2 -27640.465} C_VEL
LIN {X 0,Y 79.676,Z 673.983,A -85,B 0,C 180,E1 -27650.66,E2 -27650.66} C_VEL
LIN {X 0,Y 83.979,Z 671.595,A -85,B 0,C 180,E1 -27660.14,E2 -27660.14} C_VEL
LIN {X 0,Y 90.874,Z 667.879,A -85,B 0,C 180,E1 -27669.341,E2 -27669.341} C_VEL
LIN {X 0,Y 100.027,Z 662.607,A -85,B 0,C 180,E1 -27677.539,E2 -27677.539} C_VEL
LIN {X 0,Y 111.752,Z 655.112,A -85,B 0,C 180,E1 -27684.841,E2 -27684.841} C_VEL
LIN {X 0,Y 123.52,Z 646.615,A -85,B 0,C 180,E1 -27690.19,E2 -27690.19} C_VEL
LIN {X 0,Y 134.721,Z 637.43,A -85,B 0,C 180,E1 -27694.141,E2 -27694.141} C_VEL
LIN {X 0,Y 145.36,Z 627.539,A -85,B 0,C 180,E1 -27697.245,E2 -27697.245} C_VEL
LIN {X 0,Y 155.488,Z 616.935,A -85,B 0,C 180,E1 -27699.699,E2 -27699.699} C_VEL
LIN {X 0,Y 164.773,Z 605.84,A -85,B 0,C 180,E1 -27701.625,E2 -27701.625} C_VEL
LIN {X 0,Y 173.451,Z 593.912,A -85,B 0,C 180,E1 -27703.291,E2 -27703.291} C_VEL
LIN {X 0,Y 182.114,Z 580.202,A -85,B 0,C 180,E1 -27704.746,E2 -27704.746} C_VEL
LIN {X 0,Y 190.191,Z 565.093,A -85,B 0,C 180,E1 -27705.927,E2 -27705.927} C_VEL
LIN {X 0,Y 197.481,Z 548.227,A -85,B 0,C 180,E1 -27706.961,E2 -27706.961} C_VEL
LIN {X 0,Y 203.162,Z 531.408,A -85,B 0,C 180,E1 -27707.727,E2 -27707.727} C_VEL
LIN {X 0,Y 207.304,Z 514.949,A -85,B 0,C 180,E1 -27708.251,E2 -27708.251} C_VEL
LIN {X 0,Y 210.141,Z 498.298,A -85,B 0,C 180,E1 -27708.654,E2 -27708.654} C_VEL
LIN {X 0,Y 213.913,Z 465.161,A -85,B 0,C 180,E1 -27709.305,E2 -27709.305} C_VEL
LIN {X 0,Y 212.545,Z 461.053,A -85,B 0,C 180,E1 -27712.529,E2 -27712.529} C_VEL
LIN {X 0,Y 211.698,Z 458.375,A -85,B 0,C 180,E1 -27715.716,E2 -27715.716} C_VEL
LIN {X 0,Y 211.302,Z 457.193,A -85,B 0,C 180,E1 -27720,E2 -27720} C_VEL
LIN {X 0,Y 211.808,Z 458.729,A -85,B 0,C 180,E1 -27724.46,E2 -27724.46} C_VEL
LIN {X 0,Y 212.83,Z 462.015,A -85,B 0,C 180,E1 -27727.912,E2 -27727.912} C_VEL
LIN {X 0,Y 213.933,Z 465.198,A -85,B 0,C 180,E1 -27730.364,E2 -27730.364} C_VEL
LIN {X 0,Y 209.225,Z 505.71,A -85,B 0,C 180,E1 -27731.163,E2 -27731.163} C_VEL
LIN {X 0,Y 205.798,Z 522.868,A -85,B 0,C 180,E1 -27731.573,E2 -27731.573} C_VEL
LIN {X 0,Y 201.225,Z 538.941,A -85,B 0,C 180,E1 -27732.063,E2 -27732.063} C_VEL
LIN {X 0,Y 195.198,Z 555.286,A -85,B 0,C 180,E1 -27732.753,E2 -27732.753} C_VEL
LIN {X 0,Y 188.043,Z 570.886,A -85,B 0,C 180,E1 -27733.657,E2 -27733.657} C_VEL
LIN {X 0,Y 179.91,Z 585.617,A -85,B 0,C 180,E1 -27734.8,E2 -27734.8} C_VEL
LIN {X 0,Y 171.046,Z 599.178,A -85,B 0,C 180,E1 -27736.172,E2 -27736.172} C_VEL
LIN {X 0,Y 162.33,Z 610.706,A -85,B 0,C 180,E1 -27737.736,E2 -27737.736} C_VEL
LIN {X 0,Y 152.977,Z 621.681,A -85,B 0,C 180,E1 -27739.646,E2 -27739.646} C_VEL
LIN {X 0,Y 142.305,Z 632.633,A -85,B 0,C 180,E1 -27742.182,E2 -27742.182} C_VEL
LIN {X 0,Y 131.434,Z 642.458,A -85,B 0,C 180,E1 -27745.326,E2 -27745.326} C_VEL
LIN {X 0,Y 120.806,Z 651.111,A -85,B 0,C 180,E1 -27749.235,E2 -27749.235} C_VEL
LIN {X 0,Y 110.24,Z 658.768,A -85,B 0,C 180,E1 -27754.028,E2 -27754.028} C_VEL
LIN {X 0,Y 100.661,Z 665.026,A -85,B 0,C 180,E1 -27759.826,E2 -27759.826} C_VEL
LIN {X 0,Y 92.297,Z 670.166,A -85,B 0,C 180,E1 -27766.741,E2 -27766.741} C_VEL
LIN {X 0,Y 84.592,Z 674.725,A -85,B 0,C 180,E1 -27776.181,E2 -27776.181} C_VEL
LIN {X 0,Y 78.628,Z 678.296,A -85,B 0,C 180,E1 -27789.052,E2 -27789.052} C_VEL
LIN {X 0,Y 76.755,Z 679.733,A -85,B 0,C 180,E1 -27799.448,E2 -27799.448} C_VEL
LIN {X 0,Y 76.769,Z 680.284,A -85,B 0,C 180,E1 -27810,E2 -27810} C_VEL
LIN {X 0,Y 76.754,Z 679.714,A -85,B 0,C 180,E1 -27820.552,E2 -27820.552} C_VEL
LIN {X 0,Y 79.149,Z 677.886,A -85,B 0,C 180,E1 -27832.58,E2 -27832.58} C_VEL
LIN {X 0,Y 80.065,Z 676.949,A -85,B 0,C 180,E1 -27836.723,E2 -27836.723} C_VEL
LIN {X 0,Y 80.613,Z 675.094,A -85,B 0,C 180,E1 -27843.677,E2 -27843.677} C_VEL
LIN {X 0,Y 81.675,Z 673.366,A -85,B 0,C 180,E1 -27849.125,E2 -27849.125} C_VEL
LIN {X 0,Y 83.634,Z 671.844,A -85,B 0,C 180,E1 -27852.859,E2 -27852.859} C_VEL
LIN {X 0,Y 84.593,Z 671.271,A -85,B 0,C 180,E1 -27853.973,E2 -27853.973} C_VEL
LIN {X 0,Y 93.857,Z 666.149,A -85,B 0,C 180,E1 -27861.835,E2 -27861.835} C_VEL
LIN {X 0,Y 103.775,Z 660.079,A -85,B 0,C 180,E1 -27867.837,E2 -27867.837} C_VEL
LIN {X 0,Y 114.611,Z 652.773,A -85,B 0,C 180,E1 -27872.766,E2 -27872.766} C_VEL
LIN {X 0,Y 125.304,Z 644.711,A -85,B 0,C 180,E1 -27876.606,E2 -27876.606} C_VEL
LIN {X 0,Y 136.665,Z 635.005,A -85,B 0,C 180,E1 -27879.801,E2 -27879.801} C_VEL
LIN {X 0,Y 147.524,Z 624.474,A -85,B 0,C 180,E1 -27882.324,E2 -27882.324} C_VEL
LIN {X 0,Y 157.928,Z 613.047,A -85,B 0,C 180,E1 -27884.303,E2 -27884.303} C_VEL
LIN {X 0,Y 168.382,Z 599.742,A -85,B 0,C 180,E1 -27886.028,E2 -27886.028} C_VEL
LIN {X 0,Y 178.216,Z 584.976,A -85,B 0,C 180,E1 -27887.426,E2 -27887.426} C_VEL
LIN {X 0,Y 186.496,Z 570.143,A -85,B 0,C 180,E1 -27888.46,E2 -27888.46} C_VEL
LIN {X 0,Y 193.618,Z 554.723,A -85,B 0,C 180,E1 -27889.283,E2 -27889.283} C_VEL
LIN {X 0,Y 199.361,Z 539.349,A -85,B 0,C 180,E1 -27889.91,E2 -27889.91} C_VEL
LIN {X 0,Y 204.066,Z 523.258,A -85,B 0,C 180,E1 -27890.345,E2 -27890.345} C_VEL
LIN {X 0,Y 207.521,Z 506.362,A -85,B 0,C 180,E1 -27890.737,E2 -27890.737} C_VEL
LIN {X 0,Y 211.913,Z 469.907,A -85,B 0,C 180,E1 -27891.416,E2 -27891.416} C_VEL
LIN {X 0,Y 211.067,Z 467.275,A -85,B 0,C 180,E1 -27893.788,E2 -27893.788} C_VEL
LIN {X 0,Y 210.518,Z 465.196,A -85,B 0,C 180,E1 -27896.172,E2 -27896.172} C_VEL
LIN {X 0,Y 210.141,Z 463.99,A -85,B 0,C 180,E1 -27900,E2 -27900} C_VEL
LIN {X 0,Y 210.616,Z 465.526,A -85,B 0,C 180,E1 -27904.786,E2 -27904.786} C_VEL
LIN {X 0,Y 211.584,Z 468.943,A -85,B 0,C 180,E1 -27908.217,E2 -27908.217} C_VEL
LIN {X 0,Y 211.892,Z 469.875,A -85,B 0,C 180,E1 -27908.995,E2 -27908.995} C_VEL
LIN {X 0,Y 207.994,Z 502.751,A -85,B 0,C 180,E1 -27909.642,E2 -27909.642} C_VEL
LIN {X 0,Y 204.677,Z 519.603,A -85,B 0,C 180,E1 -27910.054,E2 -27910.054} C_VEL
LIN {X 0,Y 200.19,Z 535.678,A -85,B 0,C 180,E1 -27910.586,E2 -27910.586} C_VEL
LIN {X 0,Y 194.387,Z 551.611,A -85,B 0,C 180,E1 -27911.279,E2 -27911.279} C_VEL
LIN {X 0,Y 187.81,Z 566.264,A -85,B 0,C 180,E1 -27912.147,E2 -27912.147} C_VEL
LIN {X 0,Y 180.431,Z 579.815,A -85,B 0,C 180,E1 -27913.151,E2 -27913.151} C_VEL
LIN {X 0,Y 171.489,Z 593.786,A -85,B 0,C 180,E1 -27914.522,E2 -27914.522} C_VEL
LIN {X 0,Y 161.107,Z 607.58,A -85,B 0,C 180,E1 -27916.321,E2 -27916.321} C_VEL
LIN {X 0,Y 151.65,Z 618.496,A -85,B 0,C 180,E1 -27918.188,E2 -27918.188} C_VEL
LIN {X 0,Y 140.085,Z 630.069,A -85,B 0,C 180,E1 -27920.855,E2 -27920.855} C_VEL
LIN {X 0,Y 128.862,Z 639.82,A -85,B 0,C 180,E1 -27924.003,E2 -27924.003} C_VEL
LIN {X 0,Y 118.749,Z 647.607,A -85,B 0,C 180,E1 -27927.408,E2 -27927.408} C_VEL
LIN {X 0,Y 107.834,Z 655.13,A -85,B 0,C 180,E1 -27932.085,E2 -27932.085} C_VEL
LIN {X 0,Y 95.375,Z 662.674,A -85,B 0,C 180,E1 -27939.311,E2 -27939.311} C_VEL
LIN {X 0,Y 84.725,Z 668.39,A -85,B 0,C 180,E1 -27948.425,E2 -27948.425} C_VEL
LIN {X 0,Y 77.913,Z 671.724,A -85,B 0,C 180,E1 -27957.233,E2 -27957.233} C_VEL
LIN {X 0,Y 73.063,Z 674.138,A -85,B 0,C 180,E1 -27967.371,E2 -27967.371} C_VEL
LIN {X 0,Y 70.392,Z 675.493,A -85,B 0,C 180,E1 -27978.482,E2 -27978.482} C_VEL
LIN {X 0,Y 69.781,Z 676.005,A -85,B 0,C 180,E1 -27990,E2 -27990} C_VEL
LIN {X 0,Y 70.39,Z 675.52,A -85,B 0,C 180,E1 -28001.518,E2 -28001.518} C_VEL
LIN {X 0,Y 73.038,Z 674.191,A -85,B 0,C 180,E1 -28012.637,E2 -28012.637} C_VEL
LIN {X 0,Y 77.875,Z 671.803,A -85,B 0,C 180,E1 -28022.784,E2 -28022.784} C_VEL
LIN {X 0,Y 84.972,Z 668.347,A -85,B 0,C 180,E1 -28031.893,E2 -28031.893} C_VEL
LIN {X 0,Y 95.344,Z 662.815,A -85,B 0,C 180,E1 -28040.712,E2 -28040.712} C_VEL
LIN {X 0,Y 107.774,Z 655.321,A -85,B 0,C 180,E1 -28047.966,E2 -28047.966} C_VEL
LIN {X 0,Y 120.122,Z 646.822,A -85,B 0,C 180,E1 -28053.154,E2 -28053.154} C_VEL
LIN {X 0,Y 131.765,Z 637.636,A -85,B 0,C 180,E1 -28056.935,E2 -28056.935} C_VEL
LIN {X 0,Y 142.298,Z 628.178,A -85,B 0,C 180,E1 -28059.782,E2 -28059.782} C_VEL
LIN {X 0,Y 153.155,Z 617.141,A -85,B 0,C 180,E1 -28062.208,E2 -28062.208} C_VEL
LIN {X 0,Y 162.664,Z 606.045,A -85,B 0,C 180,E1 -28064.011,E2 -28064.011} C_VEL
LIN {X 0,Y 172.432,Z 592.817,A -85,B 0,C 180,E1 -28065.721,E2 -28065.721} C_VEL
LIN {X 0,Y 181.198,Z 578.983,A -85,B 0,C 180,E1 -28067.032,E2 -28067.032} C_VEL
LIN {X 0,Y 188.593,Z 565.295,A -85,B 0,C 180,E1 -28068.016,E2 -28068.016} C_VEL
LIN {X 0,Y 196.005,Z 548.427,A -85,B 0,C 180,E1 -28068.979,E2 -28068.979} C_VEL
LIN {X 0,Y 201.701,Z 531.835,A -85,B 0,C 180,E1 -28069.687,E2 -28069.687} C_VEL
LIN {X 0,Y 205.895,Z 515.508,A -85,B 0,C 180,E1 -28070.173,E2 -28070.173} C_VEL
LIN {X 0,Y 208.838,Z 498.665,A -85,B 0,C 180,E1 -28070.557,E2 -28070.557} C_VEL
LIN {X 0,Y 212.171,Z 470.138,A -85,B 0,C 180,E1 -28071.085,E2 -28071.085} C_VEL
LIN {X 0,Y 211.354,Z 467.559,A -85,B 0,C 180,E1 -28073.397,E2 -28073.397} C_VEL
LIN {X 0,Y 210.829,Z 465.478,A -85,B 0,C 180,E1 -28075.698,E2 -28075.698} C_VEL
LIN {X 0,Y 210.436,Z 464.253,A -85,B 0,C 180,E1 -28080,E2 -28080} C_VEL
LIN {X 0,Y 210.888,Z 465.816,A -85,B 0,C 180,E1 -28084.3,E2 -28084.3} C_VEL
LIN {X 0,Y 211.731,Z 468.737,A -85,B 0,C 180,E1 -28087.39,E2 -28087.39} C_VEL
LIN {X 0,Y 212.186,Z 470.188,A -85,B 0,C 180,E1 -28088.587,E2 -28088.587} C_VEL
LIN {X 0,Y 208.006,Z 505.243,A -85,B 0,C 180,E1 -28089.235,E2 -28089.235} C_VEL
LIN {X 0,Y 204.703,Z 521.755,A -85,B 0,C 180,E1 -28089.604,E2 -28089.604} C_VEL
LIN {X 0,Y 200.277,Z 537.438,A -85,B 0,C 180,E1 -28090.022,E2 -28090.022} C_VEL
LIN {X 0,Y 194.806,Z 552.582,A -85,B 0,C 180,E1 -28090.591,E2 -28090.591} C_VEL
LIN {X 0,Y 188.155,Z 567.458,A -85,B 0,C 180,E1 -28091.338,E2 -28091.338} C_VEL
LIN {X 0,Y 179.877,Z 582.672,A -85,B 0,C 180,E1 -28092.374,E2 -28092.374} C_VEL
LIN {X 0,Y 170.829,Z 596.618,A -85,B 0,C 180,E1 -28093.606,E2 -28093.606} C_VEL
LIN {X 0,Y 160.813,Z 609.862,A -85,B 0,C 180,E1 -28095.201,E2 -28095.201} C_VEL
LIN {X 0,Y 150.724,Z 621.474,A -85,B 0,C 180,E1 -28097.085,E2 -28097.085} C_VEL
LIN {X 0,Y 139.745,Z 632.425,A -85,B 0,C 180,E1 -28099.445,E2 -28099.445} C_VEL
LIN {X 0,Y 127.767,Z 642.875,A -85,B 0,C 180,E1 -28102.646,E2 -28102.646} C_VEL
LIN {X 0,Y 117.475,Z 650.903,A -85,B 0,C 180,E1 -28106.185,E2 -28106.185} C_VEL
LIN {X 0,Y 106.371,Z 658.558,A -85,B 0,C 180,E1 -28110.805,E2 -28110.805} C_VEL
LIN {X 0,Y 96.206,Z 664.817,A -85,B 0,C 180,E1 -28116.529,E2 -28116.529} C_VEL
LIN {X 0,Y 87.172,Z 669.956,A -85,B 0,C 180,E1 -28123.482,E2 -28123.482} C_VEL
LIN {X 0,Y 79.683,Z 673.968,A -85,B 0,C 180,E1 -28131.874,E2 -28131.874} C_VEL
LIN {X 0,Y 74.031,Z 676.944,A -85,B 0,C 180,E1 -28141.663,E2 -28141.663} C_VEL
LIN {X 0,Y 70.561,Z 678.92,A -85,B 0,C 180,E1 -28152.615,E2 -28152.615} C_VEL
LIN {X 0,Y 69.495,Z 679.912,A -85,B 0,C 180,E1 -28164.196,E2 -28164.196} C_VEL
LIN {X 0,Y 69.662,Z 680.077,A -85,B 0,C 180,E1 -28170,E2 -28170} C_VEL
LIN {X 0,Y 69.738,Z 679.505,A -85,B 0,C 180,E1 -28181.628,E2 -28181.628} C_VEL
LIN {X 0,Y 72.273,Z 677.856,A -85,B 0,C 180,E1 -28193.905,E2 -28193.905} C_VEL
LIN {X 0,Y 78.264,Z 674.683,A -85,B 0,C 180,E1 -28206.083,E2 -28206.083} C_VEL
LIN {X 0,Y 84.593,Z 671.271,A -85,B 0,C 180,E1 -28213.973,E2 -28213.973} C_VEL
LIN {X 0,Y 87.257,Z 669.587,A -85,B 0,C 180,E1 -28217.299,E2 -28217.299} C_VEL
LIN {X 0,Y 90.702,Z 666.55,A -85,B 0,C 180,E1 -28222.982,E2 -28222.982} C_VEL
LIN {X 0,Y 93.884,Z 663.898,A -85,B 0,C 180,E1 -28227.198,E2 -28227.198} C_VEL
LIN {X 0,Y 97.156,Z 661.666,A -85,B 0,C 180,E1 -28229.827,E2 -28229.827} C_VEL
LIN {X 0,Y 98.474,Z 660.844,A -85,B 0,C 180,E1 -28230.545,E2 -28230.545} C_VEL
LIN {X 0,Y 108.586,Z 654.549,A -85,B 0,C 180,E1 -28234.973,E2 -28234.973} C_VEL
LIN {X 0,Y 120.408,Z 646.139,A -85,B 0,C 180,E1 -28239.049,E2 -28239.049} C_VEL
LIN {X 0,Y 132.775,Z 636.156,A -85,B 0,C 180,E1 -28242.32,E2 -28242.32} C_VEL
LIN {X 0,Y 143.896,Z 625.898,A -85,B 0,C 180,E1 -28244.709,E2 -28244.709} C_VEL
LIN {X 0,Y 155.647,Z 613.426,A -85,B 0,C 180,E1 -28246.757,E2 -28246.757} C_VEL
LIN {X 0,Y 165.973,Z 600.61,A -85,B 0,C 180,E1 -28248.295,E2 -28248.295} C_VEL
LIN {X 0,Y 175.132,Z 587.357,A -85,B 0,C 180,E1 -28249.474,E2 -28249.474} C_VEL
LIN {X 0,Y 183.521,Z 573.104,A -85,B 0,C 180,E1 -28250.436,E2 -28250.436} C_VEL
LIN {X 0,Y 190.263,Z 559.556,A -85,B 0,C 180,E1 -28251.15,E2 -28251.15} C_VEL
LIN {X 0,Y 196.692,Z 543.628,A -85,B 0,C 180,E1 -28251.783,E2 -28251.783} C_VEL
LIN {X 0,Y 201.873,Z 527.208,A -85,B 0,C 180,E1 -28252.225,E2 -28252.225} C_VEL
LIN {X 0,Y 205.748,Z 510.223,A -85,B 0,C 180,E1 -28252.592,E2 -28252.592} C_VEL
LIN {X 0,Y 208.469,Z 491.307,A -85,B 0,C 180,E1 -28252.941,E2 -28252.941} C_VEL
LIN {X 0,Y 210.349,Z 475.065,A -85,B 0,C 180,E1 -28253.224,E2 -28253.224} C_VEL
LIN {X 0,Y 209.551,Z 472.13,A -85,B 0,C 180,E1 -28256.636,E2 -28256.636} C_VEL
LIN {X 0,Y 209.274,Z 471.046,A -85,B 0,C 180,E1 -28260,E2 -28260} C_VEL
LIN {X 0,Y 209.665,Z 472.477,A -85,B 0,C 180,E1 -28264.446,E2 -28264.446} C_VEL
LIN {X 0,Y 210.333,Z 475.073,A -85,B 0,C 180,E1 -28267.199,E2 -28267.199} C_VEL
LIN {X 0,Y 206.738,Z 504.219,A -85,B 0,C 180,E1 -28267.733,E2 -28267.733} C_VEL
LIN {X 0,Y 203.256,Z 521.154,A -85,B 0,C 180,E1 -28268.128,E2 -28268.128} C_VEL
LIN {X 0,Y 198.585,Z 537.191,A -85,B 0,C 180,E1 -28268.616,E2 -28268.616} C_VEL
LIN {X 0,Y 193.127,Z 551.824,A -85,B 0,C 180,E1 -28269.217,E2 -28269.217} C_VEL
LIN {X 0,Y 186.447,Z 566.476,A -85,B 0,C 180,E1 -28270.017,E2 -28270.017} C_VEL
LIN {X 0,Y 178.948,Z 580.027,A -85,B 0,C 180,E1 -28270.935,E2 -28270.935} C_VEL
LIN {X 0,Y 170.58,Z 592.951,A -85,B 0,C 180,E1 -28272.089,E2 -28272.089} C_VEL
LIN {X 0,Y 160.888,Z 605.85,A -85,B 0,C 180,E1 -28273.608,E2 -28273.608} C_VEL
LIN {X 0,Y 151.174,Z 616.979,A -85,B 0,C 180,E1 -28275.279,E2 -28275.279} C_VEL
LIN {X 0,Y 140.017,Z 628.08,A -85,B 0,C 180,E1 -28277.508,E2 -28277.508} C_VEL
LIN {X 0,Y 129.176,Z 637.588,A -85,B 0,C 180,E1 -28280.198,E2 -28280.198} C_VEL
LIN {X 0,Y 117.117,Z 646.815,A -85,B 0,C 180,E1 -28283.777,E2 -28283.777} C_VEL
LIN {X 0,Y 104.194,Z 655.342,A -85,B 0,C 180,E1 -28288.735,E2 -28288.735} C_VEL
LIN {X 0,Y 91.002,Z 662.884,A -85,B 0,C 180,E1 -28295.816,E2 -28295.816} C_VEL
LIN {X 0,Y 79.513,Z 668.599,A -85,B 0,C 180,E1 -28305.001,E2 -28305.001} C_VEL
LIN {X 0,Y 72.004,Z 671.933,A -85,B 0,C 180,E1 -28314.152,E2 -28314.152} C_VEL
LIN {X 0,Y 66.534,Z 674.346,A -85,B 0,C 180,E1 -28325.006,E2 -28325.006} C_VEL
LIN {X 0,Y 63.441,Z 675.701,A -85,B 0,C 180,E1 -28337.199,E2 -28337.199} C_VEL
LIN {X 0,Y 62.696,Z 676.212,A -85,B 0,C 180,E1 -28350,E2 -28350} C_VEL
LIN {X 0,Y 63.439,Z 675.727,A -85,B 0,C 180,E1 -28362.801,E2 -28362.801} C_VEL
LIN {X 0,Y 66.511,Z 674.399,A -85,B 0,C 180,E1 -28375.003,E2 -28375.003} C_VEL
LIN {X 0,Y 71.969,Z 672.011,A -85,B 0,C 180,E1 -28385.867,E2 -28385.867} C_VEL
LIN {X 0,Y 79.483,Z 668.707,A -85,B 0,C 180,E1 -28395.021,E2 -28395.021} C_VEL
LIN {X 0,Y 90.972,Z 663.023,A -85,B 0,C 180,E1 -28404.209,E2 -28404.209} C_VEL
LIN {X 0,Y 104.142,Z 655.529,A -85,B 0,C 180,E1 -28411.317,E2 -28411.317} C_VEL
LIN {X 0,Y 117.066,Z 647.029,A -85,B 0,C 180,E1 -28416.279,E2 -28416.279} C_VEL
LIN {X 0,Y 129.136,Z 637.842,A -85,B 0,C 180,E1 -28419.849,E2 -28419.849} C_VEL
LIN {X 0,Y 141.564,Z 626.91,A -85,B 0,C 180,E1 -28422.874,E2 -28422.874} C_VEL
LIN {X 0,Y 152.732,Z 615.575,A -85,B 0,C 180,E1 -28425.085,E2 -28425.085} C_VEL
LIN {X 0,Y 163.302,Z 603.213,A -85,B 0,C 180,E1 -28426.83,E2 -28426.83} C_VEL
LIN {X 0,Y 173.107,Z 589.753,A -85,B 0,C 180,E1 -28428.363,E2 -28428.363} C_VEL
LIN {X 0,Y 181.402,Z 576.344,A -85,B 0,C 180,E1 -28429.447,E2 -28429.447} C_VEL
LIN {X 0,Y 188.914,Z 561.977,A -85,B 0,C 180,E1 -28430.348,E2 -28430.348} C_VEL
LIN {X 0,Y 195.611,Z 546.377,A -85,B 0,C 180,E1 -28431.124,E2 -28431.124} C_VEL
LIN {X 0,Y 201.117,Z 530.099,A -85,B 0,C 180,E1 -28431.753,E2 -28431.753} C_VEL
LIN {X 0,Y 205.304,Z 513.519,A -85,B 0,C 180,E1 -28432.185,E2 -28432.185} C_VEL
LIN {X 0,Y 207.999,Z 497.349,A -85,B 0,C 180,E1 -28432.519,E2 -28432.519} C_VEL
LIN {X 0,Y 210.61,Z 475.33,A -85,B 0,C 180,E1 -28432.893,E2 -28432.893} C_VEL
LIN {X 0,Y 209.862,Z 472.399,A -85,B 0,C 180,E1 -28436.159,E2 -28436.159} C_VEL
LIN {X 0,Y 209.567,Z 471.33,A -85,B 0,C 180,E1 -28440,E2 -28440} C_VEL
LIN {X 0,Y 209.943,Z 472.788,A -85,B 0,C 180,E1 -28443.989,E2 -28443.989} C_VEL
LIN {X 0,Y 210.608,Z 475.338,A -85,B 0,C 180,E1 -28446.737,E2 -28446.737} C_VEL
LIN {X 0,Y 206.693,Z 506.754,A -85,B 0,C 180,E1 -28447.331,E2 -28447.331} C_VEL
LIN {X 0,Y 203.027,Z 524.129,A -85,B 0,C 180,E1 -28447.684,E2 -28447.684} C_VEL
LIN {X 0,Y 197.956,Z 540.959,A -85,B 0,C 180,E1 -28448.129,E2 -28448.129} C_VEL
LIN {X 0,Y 191.948,Z 556.305,A -85,B 0,C 180,E1 -28448.672,E2 -28448.672} C_VEL
LIN {X 0,Y 184.353,Z 572.066,A -85,B 0,C 180,E1 -28449.457,E2 -28449.457} C_VEL
LIN {X 0,Y 175.967,Z 586.504,A -85,B 0,C 180,E1 -28450.425,E2 -28450.425} C_VEL
LIN {X 0,Y 166.801,Z 599.901,A -85,B 0,C 180,E1 -28451.591,E2 -28451.591} C_VEL
LIN {X 0,Y 155.967,Z 613.405,A -85,B 0,C 180,E1 -28453.232,E2 -28453.232} C_VEL
LIN {X 0,Y 143.906,Z 626.173,A -85,B 0,C 180,E1 -28455.306,E2 -28455.306} C_VEL
LIN {X 0,Y 132.783,Z 636.381,A -85,B 0,C 180,E1 -28457.692,E2 -28457.692} C_VEL
LIN {X 0,Y 120.437,Z 646.325,A -85,B 0,C 180,E1 -28460.987,E2 -28460.987} C_VEL
LIN {X 0,Y 111.499,Z 652.727,A -85,B 0,C 180,E1 -28463.942,E2 -28463.942} C_VEL
LIN {X 0,Y 100.086,Z 659.996,A -85,B 0,C 180,E1 -28468.63,E2 -28468.63} C_VEL
LIN {X 0,Y 89.545,Z 666.042,A -85,B 0,C 180,E1 -28474.504,E2 -28474.504} C_VEL
LIN {X 0,Y 78.055,Z 671.916,A -85,B 0,C 180,E1 -28483.92,E2 -28483.92} C_VEL
LIN {X 0,Y 70.7,Z 675.361,A -85,B 0,C 180,E1 -28493.386,E2 -28493.386} C_VEL
LIN {X 0,Y 65.439,Z 677.878,A -85,B 0,C 180,E1 -28504.559,E2 -28504.559} C_VEL
LIN {X 0,Y 62.762,Z 679.316,A -85,B 0,C 180,E1 -28517.059,E2 -28517.059} C_VEL
LIN {X 0,Y 62.55,Z 679.869,A -85,B 0,C 180,E1 -28530,E2 -28530} C_VEL
LIN {X 0,Y 62.762,Z 679.296,A -85,B 0,C 180,E1 -28542.942,E2 -28542.942} C_VEL
LIN {X 0,Y 65.437,Z 677.839,A -85,B 0,C 180,E1 -28555.443,E2 -28555.443} C_VEL
LIN {X 0,Y 72.054,Z 674.69,A -85,B 0,C 180,E1 -28568.713,E2 -28568.713} C_VEL
LIN {X 0,Y 80.175,Z 670.75,A -85,B 0,C 180,E1 -28578.167,E2 -28578.167} C_VEL
LIN {X 0,Y 89.569,Z 665.937,A -85,B 0,C 180,E1 -28585.474,E2 -28585.474} C_VEL
LIN {X 0,Y 98.474,Z 660.844,A -85,B 0,C 180,E1 -28590.545,E2 -28590.545} C_VEL
LIN {X 0,Y 102.204,Z 658.44,A -85,B 0,C 180,E1 -28592.755,E2 -28592.755} C_VEL
LIN {X 0,Y 112.87,Z 649.8,A -85,B 0,C 180,E1 -28600.425,E2 -28600.425} C_VEL
LIN {X 0,Y 116.871,Z 646.759,A -85,B 0,C 180,E1 -28601.996,E2 -28601.996} C_VEL
LIN {X 0,Y 129.159,Z 637.307,A -85,B 0,C 180,E1 -28604.981,E2 -28604.981} C_VEL
LIN {X 0,Y 140.528,Z 627.272,A -85,B 0,C 180,E1 -28607.216,E2 -28607.216} C_VEL
LIN {X 0,Y 151.643,Z 615.972,A -85,B 0,C 180,E1 -28608.954,E2 -28608.954} C_VEL
LIN {X 0,Y 162.146,Z 603.616,A -85,B 0,C 180,E1 -28610.423,E2 -28610.423} C_VEL
LIN {X 0,Y 171.42,Z 591.031,A -85,B 0,C 180,E1 -28611.527,E2 -28611.527} C_VEL
LIN {X 0,Y 180.766,Z 576.036,A -85,B 0,C 180,E1 -28612.483,E2 -28612.483} C_VEL
LIN {X 0,Y 188.441,Z 561.116,A -85,B 0,C 180,E1 -28613.209,E2 -28613.209} C_VEL
LIN {X 0,Y 194.993,Z 545.526,A -85,B 0,C 180,E1 -28613.793,E2 -28613.793} C_VEL
LIN {X 0,Y 200.516,Z 528.842,A -85,B 0,C 180,E1 -28614.186,E2 -28614.186} C_VEL
LIN {X 0,Y 204.553,Z 512.131,A -85,B 0,C 180,E1 -28614.527,E2 -28614.527} C_VEL
LIN {X 0,Y 207.292,Z 494.663,A -85,B 0,C 180,E1 -28614.831,E2 -28614.831} C_VEL
LIN {X 0,Y 208.946,Z 480.568,A -85,B 0,C 180,E1 -28615.08,E2 -28615.08} C_VEL
LIN {X 0,Y 208.684,Z 479.205,A -85,B 0,C 180,E1 -28616.622,E2 -28616.622} C_VEL
LIN {X 0,Y 208.403,Z 478.137,A -85,B 0,C 180,E1 -28620,E2 -28620} C_VEL
LIN {X 0,Y 208.729,Z 479.411,A -85,B 0,C 180,E1 -28624.127,E2 -28624.127} C_VEL
LIN {X 0,Y 208.938,Z 480.585,A -85,B 0,C 180,E1 -28625.357,E2 -28625.357} C_VEL
LIN {X 0,Y 205.931,Z 504.296,A -85,B 0,C 180,E1 -28625.779,E2 -28625.779} C_VEL
LIN {X 0,Y 202.33,Z 521.567,A -85,B 0,C 180,E1 -28626.144,E2 -28626.144} C_VEL
LIN {X 0,Y 197.649,Z 537.405,A -85,B 0,C 180,E1 -28626.59,E2 -28626.59} C_VEL
LIN {X 0,Y 192.119,Z 552.037,A -85,B 0,C 180,E1 -28627.132,E2 -28627.132} C_VEL
LIN {X 0,Y 185.344,Z 566.688,A -85,B 0,C 180,E1 -28627.854,E2 -28627.854} C_VEL
LIN {X 0,Y 177.738,Z 580.239,A -85,B 0,C 180,E1 -28628.687,E2 -28628.687} C_VEL
LIN {X 0,Y 168.513,Z 594.172,A -85,B 0,C 180,E1 -28629.832,E2 -28629.832} C_VEL
LIN {X 0,Y 157.703,Z 608.001,A -85,B 0,C 180,E1 -28631.358,E2 -28631.358} C_VEL
LIN {X 0,Y 147.817,Z 618.918,A -85,B 0,C 180,E1 -28632.923,E2 -28632.923} C_VEL
LIN {X 0,Y 135.68,Z 630.45,A -85,B 0,C 180,E1 -28635.159,E2 -28635.159} C_VEL
LIN {X 0,Y 123.728,Z 640.242,A -85,B 0,C 180,E1 -28637.931,E2 -28637.931} C_VEL
LIN {X 0,Y 112.885,Z 648.028,A -85,B 0,C 180,E1 -28640.955,E2 -28640.955} C_VEL
LIN {X 0,Y 100.938,Z 655.553,A -85,B 0,C 180,E1 -28645.157,E2 -28645.157} C_VEL
LIN {X 0,Y 87.005,Z 663.094,A -85,B 0,C 180,E1 -28651.989,E2 -28651.989} C_VEL
LIN {X 0,Y 74.626,Z 668.809,A -85,B 0,C 180,E1 -28661.114,E2 -28661.114} C_VEL
LIN {X 0,Y 66.344,Z 672.142,A -85,B 0,C 180,E1 -28670.536,E2 -28670.536} C_VEL
LIN {X 0,Y 60.13,Z 674.555,A -85,B 0,C 180,E1 -28682.126,E2 -28682.126} C_VEL
LIN {X 0,Y 56.516,Z 675.909,A -85,B 0,C 180,E1 -28695.599,E2 -28695.599} C_VEL
LIN {X 0,Y 55.604,Z 676.419,A -85,B 0,C 180,E1 -28710,E2 -28710} C_VEL
LIN {X 0,Y 56.512,Z 675.935,A -85,B 0,C 180,E1 -28724.402,E2 -28724.402} C_VEL
LIN {X 0,Y 60.108,Z 674.607,A -85,B 0,C 180,E1 -28737.884,E2 -28737.884} C_VEL
LIN {X 0,Y 66.312,Z 672.219,A -85,B 0,C 180,E1 -28749.486,E2 -28749.486} C_VEL
LIN {X 0,Y 74.602,Z 668.915,A -85,B 0,C 180,E1 -28758.907,E2 -28758.907} C_VEL
LIN {X 0,Y 86.966,Z 663.232,A -85,B 0,C 180,E1 -28768.052,E2 -28768.052} C_VEL
LIN {X 0,Y 100.895,Z 655.737,A -85,B 0,C 180,E1 -28774.894,E2 -28774.894} C_VEL
LIN {X 0,Y 114.377,Z 647.237,A -85,B 0,C 180,E1 -28779.56,E2 -28779.56} C_VEL
LIN {X 0,Y 126.853,Z 638.049,A -85,B 0,C 180,E1 -28782.878,E2 -28782.878} C_VEL
LIN {X 0,Y 138.012,Z 628.591,A -85,B 0,C 180,E1 -28785.358,E2 -28785.358} C_VEL
LIN {X 0,Y 149.416,Z 617.552,A -85,B 0,C 180,E1 -28787.421,E2 -28787.421} C_VEL
LIN {X 0,Y 159.336,Z 606.454,A -85,B 0,C 180,E1 -28788.931,E2 -28788.931} C_VEL
LIN {X 0,Y 169.059,Z 593.817,A -85,B 0,C 180,E1 -28790.337,E2 -28790.337} C_VEL
LIN {X 0,Y 177.702,Z 580.811,A -85,B 0,C 180,E1 -28791.388,E2 -28791.388} C_VEL
LIN {X 0,Y 186.163,Z 565.698,A -85,B 0,C 180,E1 -28792.297,E2 -28792.297} C_VEL
LIN {X 0,Y 193.371,Z 549.86,A -85,B 0,C 180,E1 -28793.05,E2 -28793.05} C_VEL
LIN {X 0,Y 199.014,Z 534.172,A -85,B 0,C 180,E1 -28793.631,E2 -28793.631} C_VEL
LIN {X 0,Y 203.299,Z 518.712,A -85,B 0,C 180,E1 -28794.033,E2 -28794.033} C_VEL
LIN {X 0,Y 206.561,Z 502.051,A -85,B 0,C 180,E1 -28794.381,E2 -28794.381} C_VEL
LIN {X 0,Y 209.215,Z 480.847,A -85,B 0,C 180,E1 -28794.749,E2 -28794.749} C_VEL
LIN {X 0,Y 208.899,Z 479.308,A -85,B 0,C 180,E1 -28796.681,E2 -28796.681} C_VEL
LIN {X 0,Y 208.698,Z 478.404,A -85,B 0,C 180,E1 -28800,E2 -28800} C_VEL
LIN {X 0,Y 208.993,Z 479.727,A -85,B 0,C 180,E1 -28803.615,E2 -28803.615} C_VEL
LIN {X 0,Y 209.225,Z 480.917,A -85,B 0,C 180,E1 -28804.943,E2 -28804.943} C_VEL
LIN {X 0,Y 205.95,Z 506.329,A -85,B 0,C 180,E1 -28805.366,E2 -28805.366} C_VEL
LIN {X 0,Y 202.305,Z 523.534,A -85,B 0,C 180,E1 -28805.685,E2 -28805.685} C_VEL
LIN {X 0,Y 197.362,Z 539.888,A -85,B 0,C 180,E1 -28806.054,E2 -28806.054} C_VEL
LIN {X 0,Y 191.842,Z 554.175,A -85,B 0,C 180,E1 -28806.505,E2 -28806.505} C_VEL
LIN {X 0,Y 185.027,Z 568.692,A -85,B 0,C 180,E1 -28807.11,E2 -28807.11} C_VEL
LIN {X 0,Y 176.522,Z 583.69,A -85,B 0,C 180,E1 -28807.964,E2 -28807.964} C_VEL
LIN {X 0,Y 167.2,Z 597.386,A -85,B 0,C 180,E1 -28808.967,E2 -28808.967} C_VEL
LIN {X 0,Y 157.121,Z 610.088,A -85,B 0,C 180,E1 -28810.248,E2 -28810.248} C_VEL
LIN {X 0,Y 147.159,Z 621.062,A -85,B 0,C 180,E1 -28811.756,E2 -28811.756} C_VEL
LIN {X 0,Y 135.638,Z 632.01,A -85,B 0,C 180,E1 -28813.71,E2 -28813.71} C_VEL
LIN {X 0,Y 124.37,Z 641.359,A -85,B 0,C 180,E1 -28816.128,E2 -28816.128} C_VEL
LIN {X 0,Y 113.414,Z 649.469,A -85,B 0,C 180,E1 -28819.092,E2 -28819.092} C_VEL
LIN {X 0,Y 99.764,Z 658.141,A -85,B 0,C 180,E1 -28823.681,E2 -28823.681} C_VEL
LIN {X 0,Y 85.666,Z 665.832,A -85,B 0,C 180,E1 -28830.525,E2 -28830.525} C_VEL
LIN {X 0,Y 73.233,Z 671.706,A -85,B 0,C 180,E1 -28839.849,E2 -28839.849} C_VEL
LIN {X 0,Y 65.058,Z 675.152,A -85,B 0,C 180,E1 -28849.598,E2 -28849.598} C_VEL
LIN {X 0,Y 59.049,Z 677.669,A -85,B 0,C 180,E1 -28861.571,E2 -28861.571} C_VEL
LIN {X 0,Y 55.806,Z 679.107,A -85,B 0,C 180,E1 -28875.412,E2 -28875.412} C_VEL
LIN {X 0,Y 55.457,Z 679.662,A -85,B 0,C 180,E1 -28890,E2 -28890} C_VEL
LIN {X 0,Y 55.806,Z 679.087,A -85,B 0,C 180,E1 -28904.589,E2 -28904.589} C_VEL
LIN {X 0,Y 59.047,Z 677.629,A -85,B 0,C 180,E1 -28918.431,E2 -28918.431} C_VEL
LIN {X 0,Y 66.032,Z 674.694,A -85,B 0,C 180,E1 -28931.84,E2 -28931.84} C_VEL
LIN {X 0,Y 75.55,Z 670.538,A -85,B 0,C 180,E1 -28942.251,E2 -28942.251} C_VEL
LIN {X 0,Y 85.683,Z 665.725,A -85,B 0,C 180,E1 -28949.456,E2 -28949.456} C_VEL
LIN {X 0,Y 99.775,Z 657.993,A -85,B 0,C 180,E1 -28956.304,E2 -28956.304} C_VEL
LIN {X 0,Y 113.373,Z 649.293,A -85,B 0,C 180,E1 -28960.97,E2 -28960.97} C_VEL
LIN {X 0,Y 116.871,Z 646.759,A -85,B 0,C 180,E1 -28961.996,E2 -28961.996} C_VEL
LIN {X 0,Y 120.903,Z 643.665,A -85,B 0,C 180,E1 -28963.434,E2 -28963.434} C_VEL
LIN {X 0,Y 132.716,Z 632.913,A -85,B 0,C 180,E1 -28968.739,E2 -28968.739} C_VEL
LIN {X 0,Y 136.731,Z 629.195,A -85,B 0,C 180,E1 -28969.718,E2 -28969.718} C_VEL
LIN {X 0,Y 149.236,Z 617.031,A -85,B 0,C 180,E1 -28971.475,E2 -28971.475} C_VEL
LIN {X 0,Y 159.405,Z 605.55,A -85,B 0,C 180,E1 -28972.745,E2 -28972.745} C_VEL
LIN {X 0,Y 169.659,Z 592.055,A -85,B 0,C 180,E1 -28973.814,E2 -28973.814} C_VEL
LIN {X 0,Y 179.111,Z 577.258,A -85,B 0,C 180,E1 -28974.661,E2 -28974.661} C_VEL
LIN {X 0,Y 186.868,Z 562.672,A -85,B 0,C 180,E1 -28975.303,E2 -28975.303} C_VEL
LIN {X 0,Y 193.874,Z 546.563,A -85,B 0,C 180,E1 -28975.843,E2 -28975.843} C_VEL
LIN {X 0,Y 199.436,Z 530.324,A -85,B 0,C 180,E1 -28976.191,E2 -28976.191} C_VEL
LIN {X 0,Y 203.673,Z 513.637,A -85,B 0,C 180,E1 -28976.482,E2 -28976.482} C_VEL
LIN {X 0,Y 206.522,Z 496.431,A -85,B 0,C 180,E1 -28976.77,E2 -28976.77} C_VEL
LIN {X 0,Y 207.759,Z 486.175,A -85,B 0,C 180,E1 -28976.928,E2 -28976.928} C_VEL
LIN {X 0,Y 207.534,Z 485.221,A -85,B 0,C 180,E1 -28980,E2 -28980} C_VEL
LIN {X 0,Y 207.759,Z 486.139,A -85,B 0,C 180,E1 -28983.504,E2 -28983.504} C_VEL
LIN {X 0,Y 205.145,Z 505.549,A -85,B 0,C 180,E1 -28983.824,E2 -28983.824} C_VEL
LIN {X 0,Y 201.579,Z 522.274,A -85,B 0,C 180,E1 -28984.155,E2 -28984.155} C_VEL
LIN {X 0,Y 196.529,Z 538.918,A -85,B 0,C 180,E1 -28984.57,E2 -28984.57} C_VEL
LIN {X 0,Y 190.508,Z 554.231,A -85,B 0,C 180,E1 -28985.096,E2 -28985.096} C_VEL
LIN {X 0,Y 182.793,Z 570.055,A -85,B 0,C 180,E1 -28985.827,E2 -28985.827} C_VEL
LIN {X 0,Y 174.239,Z 584.514,A -85,B 0,C 180,E1 -28986.668,E2 -28986.668} C_VEL
LIN {X 0,Y 164.585,Z 598.282,A -85,B 0,C 180,E1 -28987.779,E2 -28987.779} C_VEL
LIN {X 0,Y 154.768,Z 610.153,A -85,B 0,C 180,E1 -28989.012,E2 -28989.012} C_VEL
LIN {X 0,Y 144.72,Z 620.746,A -85,B 0,C 180,E1 -28990.458,E2 -28990.458} C_VEL
LIN {X 0,Y 133.424,Z 631.155,A -85,B 0,C 180,E1 -28992.313,E2 -28992.313} C_VEL
LIN {X 0,Y 121.717,Z 640.453,A -85,B 0,C 180,E1 -28994.727,E2 -28994.727} C_VEL
LIN {X 0,Y 110.528,Z 648.238,A -85,B 0,C 180,E1 -28997.488,E2 -28997.488} C_VEL
LIN {X 0,Y 98.102,Z 655.764,A -85,B 0,C 180,E1 -29001.36,E2 -29001.36} C_VEL
LIN {X 0,Y 83.426,Z 663.305,A -85,B 0,C 180,E1 -29007.805,E2 -29007.805} C_VEL
LIN {X 0,Y 70.124,Z 669.019,A -85,B 0,C 180,E1 -29016.7,E2 -29016.7} C_VEL
LIN {X 0,Y 61,Z 672.351,A -85,B 0,C 180,E1 -29026.268,E2 -29026.268} C_VEL
LIN {X 0,Y 53.921,Z 674.764,A -85,B 0,C 180,E1 -29038.577,E2 -29038.577} C_VEL
LIN {X 0,Y 49.657,Z 676.117,A -85,B 0,C 180,E1 -29053.557,E2 -29053.557} C_VEL
LIN {X 0,Y 48.503,Z 676.627,A -85,B 0,C 180,E1 -29070,E2 -29070} C_VEL
LIN {X 0,Y 49.654,Z 676.142,A -85,B 0,C 180,E1 -29086.444,E2 -29086.444} C_VEL
LIN {X 0,Y 53.882,Z 674.816,A -85,B 0,C 180,E1 -29101.448,E2 -29101.448} C_VEL
LIN {X 0,Y 60.971,Z 672.427,A -85,B 0,C 180,E1 -29113.756,E2 -29113.756} C_VEL
LIN {X 0,Y 70.092,Z 669.124,A -85,B 0,C 180,E1 -29123.334,E2 -29123.334} C_VEL
LIN {X 0,Y 83.394,Z 663.44,A -85,B 0,C 180,E1 -29132.236,E2 -29132.236} C_VEL
LIN {X 0,Y 98.071,Z 655.945,A -85,B 0,C 180,E1 -29138.686,E2 -29138.686} C_VEL
LIN {X 0,Y 112.08,Z 647.444,A -85,B 0,C 180,E1 -29142.987,E2 -29142.987} C_VEL
LIN {X 0,Y 124.932,Z 638.256,A -85,B 0,C 180,E1 -29146.02,E2 -29146.02} C_VEL
LIN {X 0,Y 136.382,Z 628.797,A -85,B 0,C 180,E1 -29148.262,E2 -29148.262} C_VEL
LIN {X 0,Y 148.026,Z 617.757,A -85,B 0,C 180,E1 -29150.118,E2 -29150.118} C_VEL
LIN {X 0,Y 158.125,Z 606.658,A -85,B 0,C 180,E1 -29151.459,E2 -29151.459} C_VEL
LIN {X 0,Y 168.006,Z 594.027,A -85,B 0,C 180,E1 -29152.73,E2 -29152.73} C_VEL
LIN {X 0,Y 176.778,Z 581.013,A -85,B 0,C 180,E1 -29153.665,E2 -29153.665} C_VEL
LIN {X 0,Y 185.346,Z 565.899,A -85,B 0,C 180,E1 -29154.467,E2 -29154.467} C_VEL
LIN {X 0,Y 192.64,Z 550.061,A -85,B 0,C 180,E1 -29155.152,E2 -29155.152} C_VEL
LIN {X 0,Y 198.251,Z 534.675,A -85,B 0,C 180,E1 -29155.659,E2 -29155.659} C_VEL
LIN {X 0,Y 202.745,Z 518.652,A -85,B 0,C 180,E1 -29156.031,E2 -29156.031} C_VEL
LIN {X 0,Y 205.988,Z 502.238,A -85,B 0,C 180,E1 -29156.345,E2 -29156.345} C_VEL
LIN {X 0,Y 208.036,Z 486.445,A -85,B 0,C 180,E1 -29156.609,E2 -29156.609} C_VEL
LIN {X 0,Y 207.831,Z 485.469,A -85,B 0,C 180,E1 -29160,E2 -29160} C_VEL
LIN {X 0,Y 208.041,Z 486.471,A -85,B 0,C 180,E1 -29163.065,E2 -29163.065} C_VEL
LIN {X 0,Y 205.055,Z 507.999,A -85,B 0,C 180,E1 -29163.425,E2 -29163.425} C_VEL
LIN {X 0,Y 201.34,Z 524.728,A -85,B 0,C 180,E1 -29163.702,E2 -29163.702} C_VEL
LIN {X 0,Y 196.599,Z 540.109,A -85,B 0,C 180,E1 -29164.006,E2 -29164.006} C_VEL
LIN {X 0,Y 190.324,Z 555.903,A -85,B 0,C 180,E1 -29164.435,E2 -29164.435} C_VEL
LIN {X 0,Y 182.555,Z 571.66,A -85,B 0,C 180,E1 -29165.044,E2 -29165.044} C_VEL
LIN {X 0,Y 173.955,Z 586.096,A -85,B 0,C 180,E1 -29165.806,E2 -29165.806} C_VEL
LIN {X 0,Y 164.527,Z 599.491,A -85,B 0,C 180,E1 -29166.713,E2 -29166.713} C_VEL
LIN {X 0,Y 152.974,Z 613.374,A -85,B 0,C 180,E1 -29168.03,E2 -29168.03} C_VEL
LIN {X 0,Y 140.806,Z 625.76,A -85,B 0,C 180,E1 -29169.679,E2 -29169.679} C_VEL
LIN {X 0,Y 129.145,Z 635.966,A -85,B 0,C 180,E1 -29171.61,E2 -29171.61} C_VEL
LIN {X 0,Y 116.055,Z 645.908,A -85,B 0,C 180,E1 -29174.325,E2 -29174.325} C_VEL
LIN {X 0,Y 106.484,Z 652.311,A -85,B 0,C 180,E1 -29176.863,E2 -29176.863} C_VEL
LIN {X 0,Y 94.036,Z 659.578,A -85,B 0,C 180,E1 -29180.9,E2 -29180.9} C_VEL
LIN {X 0,Y 82.24,Z 665.623,A -85,B 0,C 180,E1 -29186.195,E2 -29186.195} C_VEL
LIN {X 0,Y 68.841,Z 671.496,A -85,B 0,C 180,E1 -29195.243,E2 -29195.243} C_VEL
LIN {X 0,Y 59.759,Z 674.942,A -85,B 0,C 180,E1 -29205.12,E2 -29205.12} C_VEL
LIN {X 0,Y 52.835,Z 677.46,A -85,B 0,C 180,E1 -29217.855,E2 -29217.855} C_VEL
LIN {X 0,Y 48.919,Z 678.898,A -85,B 0,C 180,E1 -29233.302,E2 -29233.302} C_VEL
LIN {X 0,Y 48.348,Z 679.455,A -85,B 0,C 180,E1 -29250,E2 -29250} C_VEL
LIN {X 0,Y 48.918,Z 678.878,A -85,B 0,C 180,E1 -29266.699,E2 -29266.699} C_VEL
LIN {X 0,Y 52.833,Z 677.419,A -85,B 0,C 180,E1 -29282.147,E2 -29282.147} C_VEL
LIN {X 0,Y 60.241,Z 674.7,A -85,B 0,C 180,E1 -29295.575,E2 -29295.575} C_VEL
LIN {X 0,Y 71.367,Z 670.327,A -85,B 0,C 180,E1 -29306.83,E2 -29306.83} C_VEL
LIN {X 0,Y 82.251,Z 665.513,A -85,B 0,C 180,E1 -29313.79,E2 -29313.79} C_VEL
LIN {X 0,Y 97.102,Z 657.781,A -85,B 0,C 180,E1 -29320.203,E2 -29320.203} C_VEL
LIN {X 0,Y 111.232,Z 649.081,A -85,B 0,C 180,E1 -29324.479,E2 -29324.479} C_VEL
LIN {X 0,Y 122.555,Z 640.938,A -85,B 0,C 180,E1 -29327.127,E2 -29327.127} C_VEL
LIN {X 0,Y 135.778,Z 630.05,A -85,B 0,C 180,E1 -29329.561,E2 -29329.561} C_VEL
LIN {X 0,Y 136.731,Z 629.195,A -85,B 0,C 180,E1 -29329.718,E2 -29329.718} C_VEL
LIN {X 0,Y 140.714,Z 625.442,A -85,B 0,C 180,E1 -29330.627,E2 -29330.627} C_VEL
LIN {X 0,Y 152.379,Z 612.646,A -85,B 0,C 180,E1 -29334.415,E2 -29334.415} C_VEL
LIN {X 0,Y 156.074,Z 608.346,A -85,B 0,C 180,E1 -29335.052,E2 -29335.052} C_VEL
LIN {X 0,Y 166.443,Z 595.376,A -85,B 0,C 180,E1 -29335.991,E2 -29335.991} C_VEL
LIN {X 0,Y 175.981,Z 581.337,A -85,B 0,C 180,E1 -29336.754,E2 -29336.754} C_VEL
LIN {X 0,Y 183.808,Z 567.704,A -85,B 0,C 180,E1 -29337.305,E2 -29337.305} C_VEL
LIN {X 0,Y 190.602,Z 553.389,A -85,B 0,C 180,E1 -29337.734,E2 -29337.734} C_VEL
LIN {X 0,Y 196.538,Z 538.034,A -85,B 0,C 180,E1 -29338.106,E2 -29338.106} C_VEL
LIN {X 0,Y 201.38,Z 521.879,A -85,B 0,C 180,E1 -29338.343,E2 -29338.343} C_VEL
LIN {X 0,Y 204.995,Z 504.814,A -85,B 0,C 180,E1 -29338.608,E2 -29338.608} C_VEL
LIN {X 0,Y 206.68,Z 492.665,A -85,B 0,C 180,E1 -29338.819,E2 -29338.819} C_VEL
LIN {X 0,Y 206.664,Z 492.3,A -85,B 0,C 180,E1 -29340,E2 -29340} C_VEL
LIN {X 0,Y 206.682,Z 492.651,A -85,B 0,C 180,E1 -29341.634,E2 -29341.634} C_VEL
LIN {X 0,Y 203.924,Z 510.324,A -85,B 0,C 180,E1 -29341.914,E2 -29341.914} C_VEL
LIN {X 0,Y 199.883,Z 527.121,A -85,B 0,C 180,E1 -29342.221,E2 -29342.221} C_VEL
LIN {X 0,Y 194.789,Z 542.731,A -85,B 0,C 180,E1 -29342.613,E2 -29342.613} C_VEL
LIN {X 0,Y 188.277,Z 558.371,A -85,B 0,C 180,E1 -29343.12,E2 -29343.12} C_VEL
LIN {X 0,Y 180.477,Z 573.422,A -85,B 0,C 180,E1 -29343.745,E2 -29343.745} C_VEL
LIN {X 0,Y 171.835,Z 587.295,A -85,B 0,C 180,E1 -29344.495,E2 -29344.495} C_VEL
LIN {X 0,Y 161.521,Z 601.284,A -85,B 0,C 180,E1 -29345.547,E2 -29345.547} C_VEL
LIN {X 0,Y 152.1,Z 612.293,A -85,B 0,C 180,E1 -29346.571,E2 -29346.571} C_VEL
LIN {X 0,Y 140.208,Z 624.191,A -85,B 0,C 180,E1 -29348.122,E2 -29348.122} C_VEL
LIN {X 0,Y 129.952,Z 633.086,A -85,B 0,C 180,E1 -29349.658,E2 -29349.658} C_VEL
LIN {X 0,Y 118.443,Z 641.885,A -85,B 0,C 180,E1 -29351.75,E2 -29351.75} C_VEL
LIN {X 0,Y 105.346,Z 650.445,A -85,B 0,C 180,E1 -29354.684,E2 -29354.684} C_VEL
LIN {X 0,Y 92.592,Z 657.597,A -85,B 0,C 180,E1 -29358.418,E2 -29358.418} C_VEL
LIN {X 0,Y 80.335,Z 663.515,A -85,B 0,C 180,E1 -29363.281,E2 -29363.281} C_VEL
LIN {X 0,Y 66.096,Z 669.229,A -85,B 0,C 180,E1 -29371.719,E2 -29371.719} C_VEL
LIN {X 0,Y 56.048,Z 672.561,A -85,B 0,C 180,E1 -29381.205,E2 -29381.205} C_VEL
LIN {X 0,Y 47.956,Z 674.974,A -85,B 0,C 180,E1 -29394.112,E2 -29394.112} C_VEL
LIN {X 0,Y 42.868,Z 676.325,A -85,B 0,C 180,E1 -29410.859,E2 -29410.859} C_VEL
LIN {X 0,Y 41.42,Z 676.833,A -85,B 0,C 180,E1 -29430,E2 -29430} C_VEL
LIN {X 0,Y 42.864,Z 676.35,A -85,B 0,C 180,E1 -29449.142,E2 -29449.142} C_VEL
LIN {X 0,Y 47.92,Z 675.024,A -85,B 0,C 180,E1 -29465.918,E2 -29465.918} C_VEL
LIN {X 0,Y 56.023,Z 672.635,A -85,B 0,C 180,E1 -29478.823,E2 -29478.823} C_VEL
LIN {X 0,Y 66.067,Z 669.332,A -85,B 0,C 180,E1 -29488.322,E2 -29488.322} C_VEL
LIN {X 0,Y 80.309,Z 663.648,A -85,B 0,C 180,E1 -29496.761,E2 -29496.761} C_VEL
LIN {X 0,Y 95.701,Z 656.152,A -85,B 0,C 180,E1 -29502.682,E2 -29502.682} C_VEL
LIN {X 0,Y 110.202,Z 647.651,A -85,B 0,C 180,E1 -29506.541,E2 -29506.541} C_VEL
LIN {X 0,Y 123.402,Z 638.462,A -85,B 0,C 180,E1 -29509.238,E2 -29509.238} C_VEL
LIN {X 0,Y 135.111,Z 629.003,A -85,B 0,C 180,E1 -29511.228,E2 -29511.228} C_VEL
LIN {X 0,Y 146.971,Z 617.962,A -85,B 0,C 180,E1 -29512.854,E2 -29512.854} C_VEL
LIN {X 0,Y 157.227,Z 606.863,A -85,B 0,C 180,E1 -29514.021,E2 -29514.021} C_VEL
LIN {X 0,Y 166.851,Z 594.779,A -85,B 0,C 180,E1 -29515.107,E2 -29515.107} C_VEL
LIN {X 0,Y 176.135,Z 581.216,A -85,B 0,C 180,E1 -29515.964,E2 -29515.964} C_VEL
LIN {X 0,Y 184.798,Z 566.101,A -85,B 0,C 180,E1 -29516.656,E2 -29516.656} C_VEL
LIN {X 0,Y 192.17,Z 550.262,A -85,B 0,C 180,E1 -29517.257,E2 -29517.257} C_VEL
LIN {X 0,Y 197.765,Z 535.1,A -85,B 0,C 180,E1 -29517.702,E2 -29517.702} C_VEL
LIN {X 0,Y 202.273,Z 519.29,A -85,B 0,C 180,E1 -29518.026,E2 -29518.026} C_VEL
LIN {X 0,Y 205.531,Z 503.3,A -85,B 0,C 180,E1 -29518.303,E2 -29518.303} C_VEL
LIN {X 0,Y 206.968,Z 492.938,A -85,B 0,C 180,E1 -29518.491,E2 -29518.491} C_VEL
LIN {X 0,Y 206.963,Z 492.535,A -85,B 0,C 180,E1 -29520,E2 -29520} C_VEL
LIN {X 0,Y 206.973,Z 492.925,A -85,B 0,C 180,E1 -29521.189,E2 -29521.189} C_VEL
LIN {X 0,Y 204.287,Z 510.245,A -85,B 0,C 180,E1 -29521.464,E2 -29521.464} C_VEL
LIN {X 0,Y 200.135,Z 527.577,A -85,B 0,C 180,E1 -29521.731,E2 -29521.731} C_VEL
LIN {X 0,Y 195.003,Z 543.273,A -85,B 0,C 180,E1 -29522.018,E2 -29522.018} C_VEL
LIN {X 0,Y 189.035,Z 557.691,A -85,B 0,C 180,E1 -29522.354,E2 -29522.354} C_VEL
LIN {X 0,Y 181.196,Z 573.043,A -85,B 0,C 180,E1 -29522.868,E2 -29522.868} C_VEL
LIN {X 0,Y 172.509,Z 587.187,A -85,B 0,C 180,E1 -29523.516,E2 -29523.516} C_VEL
LIN {X 0,Y 162.114,Z 601.43,A -85,B 0,C 180,E1 -29524.373,E2 -29524.373} C_VEL
LIN {X 0,Y 151.435,Z 613.909,A -85,B 0,C 180,E1 -29525.434,E2 -29525.434} C_VEL
LIN {X 0,Y 139.783,Z 625.555,A -85,B 0,C 180,E1 -29526.793,E2 -29526.793} C_VEL
LIN {X 0,Y 127.893,Z 635.759,A -85,B 0,C 180,E1 -29528.457,E2 -29528.457} C_VEL
LIN {X 0,Y 114.488,Z 645.699,A -85,B 0,C 180,E1 -29530.836,E2 -29530.836} C_VEL
LIN {X 0,Y 101.349,Z 654.07,A -85,B 0,C 180,E1 -29533.878,E2 -29533.878} C_VEL
LIN {X 0,Y 88.555,Z 660.999,A -85,B 0,C 180,E1 -29537.758,E2 -29537.758} C_VEL
LIN {X 0,Y 76.319,Z 666.68,A -85,B 0,C 180,E1 -29542.947,E2 -29542.947} C_VEL
LIN {X 0,Y 64.937,Z 671.286,A -85,B 0,C 180,E1 -29550.024,E2 -29550.024} C_VEL
LIN {X 0,Y 54.763,Z 674.766,A -85,B 0,C 180,E1 -29559.915,E2 -29559.915} C_VEL
LIN {X 0,Y 46.908,Z 677.25,A -85,B 0,C 180,E1 -29573.181,E2 -29573.181} C_VEL
LIN {X 0,Y 42.111,Z 678.689,A -85,B 0,C 180,E1 -29590.502,E2 -29590.502} C_VEL
LIN {X 0,Y 41.236,Z 679.247,A -85,B 0,C 180,E1 -29610,E2 -29610} C_VEL
LIN {X 0,Y 42.11,Z 678.669,A -85,B 0,C 180,E1 -29629.499,E2 -29629.499} C_VEL
LIN {X 0,Y 46.906,Z 677.209,A -85,B 0,C 180,E1 -29646.822,E2 -29646.822} C_VEL
LIN {X 0,Y 54.87,Z 674.67,A -85,B 0,C 180,E1 -29660.22,E2 -29660.22} C_VEL
LIN {X 0,Y 64.942,Z 671.2,A -85,B 0,C 180,E1 -29669.969,E2 -29669.969} C_VEL
LIN {X 0,Y 79.33,Z 665.302,A -85,B 0,C 180,E1 -29678.468,E2 -29678.468} C_VEL
LIN {X 0,Y 94.903,Z 657.569,A -85,B 0,C 180,E1 -29684.303,E2 -29684.303} C_VEL
LIN {X 0,Y 109.522,Z 648.869,A -85,B 0,C 180,E1 -29688.12,E2 -29688.12} C_VEL
LIN {X 0,Y 122.834,Z 639.486,A -85,B 0,C 180,E1 -29690.737,E2 -29690.737} C_VEL
LIN {X 0,Y 134.809,Z 629.707,A -85,B 0,C 180,E1 -29692.594,E2 -29692.594} C_VEL
LIN {X 0,Y 146.629,Z 618.61,A -85,B 0,C 180,E1 -29694.015,E2 -29694.015} C_VEL
LIN {X 0,Y 156.074,Z 608.346,A -85,B 0,C 180,E1 -29695.052,E2 -29695.052} C_VEL
LIN {X 0,Y 159.712,Z 603.992,A -85,B 0,C 180,E1 -29695.655,E2 -29695.655} C_VEL
LIN {X 0,Y 170.268,Z 589.465,A -85,B 0,C 180,E1 -29698.525,E2 -29698.525} C_VEL
LIN {X 0,Y 173.499,Z 584.611,A -85,B 0,C 180,E1 -29698.941,E2 -29698.941} C_VEL
LIN {X 0,Y 181.857,Z 570.665,A -85,B 0,C 180,E1 -29699.428,E2 -29699.428} C_VEL
LIN {X 0,Y 189.755,Z 554.755,A -85,B 0,C 180,E1 -29699.849,E2 -29699.849} C_VEL
LIN {X 0,Y 195.905,Z 539.378,A -85,B 0,C 180,E1 -29700.149,E2 -29700.149} C_VEL
LIN {X 0,Y 196.784,Z 536.776,A -85,B 0,C 180,E1 -29700.184,E2 -29700.184} C_VEL
LIN {X 0,Y 196.787,Z 536.755,A -85,B 0,C 180,E1 -29700.387,E2 -29700.387} C_VEL
LIN {X 0,Y 190.713,Z 552.536,A -85,B 0,C 180,E1 -29700.774,E2 -29700.774} C_VEL
LIN {X 0,Y 183.65,Z 567.325,A -85,B 0,C 180,E1 -29701.262,E2 -29701.262} C_VEL
LIN {X 0,Y 174.913,Z 582.296,A -85,B 0,C 180,E1 -29701.87,E2 -29701.87} C_VEL
LIN {X 0,Y 165.291,Z 596.032,A -85,B 0,C 180,E1 -29702.639,E2 -29702.639} C_VEL
LIN {X 0,Y 154.917,Z 608.635,A -85,B 0,C 180,E1 -29703.577,E2 -29703.577} C_VEL
LIN {X 0,Y 144.543,Z 619.551,A -85,B 0,C 180,E1 -29704.623,E2 -29704.623} C_VEL
LIN {X 0,Y 132.784,Z 630.16,A -85,B 0,C 180,E1 -29706,E2 -29706} C_VEL
LIN {X 0,Y 120.585,Z 639.653,A -85,B 0,C 180,E1 -29707.778,E2 -29707.778} C_VEL
LIN {X 0,Y 107.103,Z 648.659,A -85,B 0,C 180,E1 -29710.174,E2 -29710.174} C_VEL
LIN {X 0,Y 93.834,Z 656.186,A -85,B 0,C 180,E1 -29713.176,E2 -29713.176} C_VEL
LIN {X 0,Y 77.776,Z 663.726,A -85,B 0,C 180,E1 -29718.414,E2 -29718.414} C_VEL
LIN {X 0,Y 62.622,Z 669.439,A -85,B 0,C 180,E1 -29726.126,E2 -29726.126} C_VEL
LIN {X 0,Y 51.609,Z 672.771,A -85,B 0,C 180,E1 -29735.207,E2 -29735.207} C_VEL
LIN {X 0,Y 42.366,Z 675.183,A -85,B 0,C 180,E1 -29748.428,E2 -29748.428} C_VEL
LIN {X 0,Y 36.222,Z 676.533,A -85,B 0,C 180,E1 -29767.166,E2 -29767.166} C_VEL
LIN {X 0,Y 34.321,Z 677.041,A -85,B 0,C 180,E1 -29790,E2 -29790} C_VEL
LIN {X 0,Y 36.217,Z 676.558,A -85,B 0,C 180,E1 -29812.836,E2 -29812.836} C_VEL
LIN {X 0,Y 42.334,Z 675.233,A -85,B 0,C 180,E1 -29831.609,E2 -29831.609} C_VEL
LIN {X 0,Y 51.587,Z 672.844,A -85,B 0,C 180,E1 -29844.826,E2 -29844.826} C_VEL
LIN {X 0,Y 62.6,Z 669.54,A -85,B 0,C 180,E1 -29853.914,E2 -29853.914} C_VEL
LIN {X 0,Y 77.755,Z 663.857,A -85,B 0,C 180,E1 -29861.632,E2 -29861.632} C_VEL
LIN {X 0,Y 93.822,Z 656.36,A -85,B 0,C 180,E1 -29866.852,E2 -29866.852} C_VEL
LIN {X 0,Y 108.757,Z 647.859,A -85,B 0,C 180,E1 -29870.219,E2 -29870.219} C_VEL
LIN {X 0,Y 122.271,Z 638.669,A -85,B 0,C 180,E1 -29872.525,E2 -29872.525} C_VEL
LIN {X 0,Y 134.207,Z 629.209,A -85,B 0,C 180,E1 -29874.246,E2 -29874.246} C_VEL
LIN {X 0,Y 146.255,Z 618.168,A -85,B 0,C 180,E1 -29875.63,E2 -29875.63} C_VEL
LIN {X 0,Y 158.379,Z 605.094,A -85,B 0,C 180,E1 -29876.779,E2 -29876.779} C_VEL
LIN {X 0,Y 168.8,Z 591.757,A -85,B 0,C 180,E1 -29877.756,E2 -29877.756} C_VEL
LIN {X 0,Y 177.525,Z 578.576,A -85,B 0,C 180,E1 -29878.387,E2 -29878.387} C_VEL
LIN {X 0,Y 185.394,Z 564.543,A -85,B 0,C 180,E1 -29878.929,E2 -29878.929} C_VEL
LIN {X 0,Y 192.445,Z 549.312,A -85,B 0,C 180,E1 -29879.4,E2 -29879.4} C_VEL
LIN {X 0,Y 196.784,Z 537.734,A -85,B 0,C 180,E1 -29879.713,E2 -29879.713} C_VEL
LIN {X 0,Y 196.783,Z 537.744,A -85,B 0,C 180,E1 -29879.821,E2 -29879.821} C_VEL
LIN {X 0,Y 190.37,Z 554.106,A -85,B 0,C 180,E1 -29880.127,E2 -29880.127} C_VEL
LIN {X 0,Y 182.734,Z 569.669,A -85,B 0,C 180,E1 -29880.529,E2 -29880.529} C_VEL
LIN {X 0,Y 174.847,Z 583.078,A -85,B 0,C 180,E1 -29881.007,E2 -29881.007} C_VEL
LIN {X 0,Y 165.222,Z 596.773,A -85,B 0,C 180,E1 -29881.622,E2 -29881.622} C_VEL
LIN {X 0,Y 154.752,Z 609.471,A -85,B 0,C 180,E1 -29882.413,E2 -29882.413} C_VEL
LIN {X 0,Y 144.323,Z 620.443,A -85,B 0,C 180,E1 -29883.376,E2 -29883.376} C_VEL
LIN {X 0,Y 132.201,Z 631.389,A -85,B 0,C 180,E1 -29884.607,E2 -29884.607} C_VEL
LIN {X 0,Y 120.173,Z 640.734,A -85,B 0,C 180,E1 -29886.18,E2 -29886.18} C_VEL
LIN {X 0,Y 106.598,Z 649.859,A -85,B 0,C 180,E1 -29888.531,E2 -29888.531} C_VEL
LIN {X 0,Y 93.207,Z 657.514,A -85,B 0,C 180,E1 -29891.418,E2 -29891.418} C_VEL
LIN {X 0,Y 76.973,Z 665.204,A -85,B 0,C 180,E1 -29896.526,E2 -29896.526} C_VEL
LIN {X 0,Y 61.645,Z 671.076,A -85,B 0,C 180,E1 -29904.21,E2 -29904.21} C_VEL
LIN {X 0,Y 49.683,Z 674.776,A -85,B 0,C 180,E1 -29914.458,E2 -29914.458} C_VEL
LIN {X 0,Y 41.386,Z 677.041,A -85,B 0,C 180,E1 -29927.215,E2 -29927.215} C_VEL
LIN {X 0,Y 35.426,Z 678.48,A -85,B 0,C 180,E1 -29946.625,E2 -29946.625} C_VEL
LIN {X 0,Y 34.11,Z 679.039,A -85,B 0,C 180,E1 -29970.001,E2 -29970.001} C_VEL
LIN {X 0,Y 35.426,Z 678.459,A -85,B 0,C 180,E1 -29993.377,E2 -29993.377} C_VEL
LIN {X 0,Y 41.385,Z 676.999,A -85,B 0,C 180,E1 -30012.788,E2 -30012.788} C_VEL
LIN {X 0,Y 50.57,Z 674.459,A -85,B 0,C 180,E1 -30026.497,E2 -30026.497} C_VEL
LIN {X 0,Y 61.65,Z 670.989,A -85,B 0,C 180,E1 -30035.781,E2 -30035.781} C_VEL
LIN {X 0,Y 76.976,Z 665.09,A -85,B 0,C 180,E1 -30043.466,E2 -30043.466} C_VEL
LIN {X 0,Y 93.212,Z 657.357,A -85,B 0,C 180,E1 -30048.571,E2 -30048.571} C_VEL
LIN {X 0,Y 108.266,Z 648.656,A -85,B 0,C 180,E1 -30051.866,E2 -30051.866} C_VEL
LIN {X 0,Y 121.883,Z 639.273,A -85,B 0,C 180,E1 -30054.077,E2 -30054.077} C_VEL
LIN {X 0,Y 133.922,Z 629.626,A -85,B 0,C 180,E1 -30055.623,E2 -30055.623} C_VEL
LIN {X 0,Y 146.057,Z 618.398,A -85,B 0,C 180,E1 -30056.808,E2 -30056.808} C_VEL
LIN {X 0,Y 156.493,Z 607.154,A -85,B 0,C 180,E1 -30057.746,E2 -30057.746} C_VEL
LIN {X 0,Y 166.969,Z 593.985,A -85,B 0,C 180,E1 -30058.523,E2 -30058.523} C_VEL
LIN {X 0,Y 173.499,Z 584.611,A -85,B 0,C 180,E1 -30058.941,E2 -30058.941} C_VEL
LIN {X 0,Y 172.74,Z 585.704,A -85,B 0,C 180,E1 -30059.258,E2 -30059.258} C_VEL
LIN {X 0,Y 168.248,Z 592.096,A -85,B 0,C 180,E1 -30059.787,E2 -30059.787} C_VEL
LIN {X 0,Y 160.66,Z 601.859,A -85,B 0,C 180,E1 -30060.184,E2 -30060.184} C_VEL
LIN {X 0,Y 154.679,Z 608.856,A -85,B 0,C 180,E1 -30060.215,E2 -30060.215} C_VEL
LIN {X 0,Y 152.64,Z 611.102,A -85,B 0,C 180,E1 -30060.127,E2 -30060.127} C_VEL
LIN {X 0,Y 140.572,Z 623.205,A -85,B 0,C 180,E1 -30059.235,E2 -30059.235} C_VEL
LIN {X 0,Y 128.324,Z 633.733,A -85,B 0,C 180,E1 -30058.186,E2 -30058.186} C_VEL
LIN {X 0,Y 116.139,Z 642.785,A -85,B 0,C 180,E1 -30056.826,E2 -30056.826} C_VEL
LIN {X 0,Y 104.04,Z 650.483,A -85,B 0,C 180,E1 -30055.117,E2 -30055.117} C_VEL
LIN {X 0,Y 92.055,Z 657.145,A -85,B 0,C 180,E1 -30052.974,E2 -30052.974} C_VEL
LIN {X 0,Y 75.15,Z 664.917,A -85,B 0,C 180,E1 -30048.715,E2 -30048.715} C_VEL
LIN {X 0,Y 59.055,Z 670.777,A -85,B 0,C 180,E1 -30042.185,E2 -30042.185} C_VEL
LIN {X 0,Y 45.283,Z 674.691,A -85,B 0,C 180,E1 -30032.253,E2 -30032.253} C_VEL
LIN {X 0,Y 36.448,Z 676.789,A -85,B 0,C 180,E1 -30020.469,E2 -30020.469} C_VEL
LIN {X 0,Y 28.988,Z 678.25,A -85,B 0,C 180,E1 -29999.006,E2 -29999.006} C_VEL
LIN {X 0,Y 26.999,Z 678.831,A -85,B 0,C 180,E1 -29970.001,E2 -29970.001} C_VEL
LIN {X 0,Y 28.988,Z 678.271,A -85,B 0,C 180,E1 -29940.996,E2 -29940.996} C_VEL
LIN {X 0,Y 36.449,Z 676.832,A -85,B 0,C 180,E1 -29919.534,E2 -29919.534} C_VEL
LIN {X 0,Y 46.972,Z 674.312,A -85,B 0,C 180,E1 -29906.141,E2 -29906.141} C_VEL
LIN {X 0,Y 59.051,Z 670.866,A -85,B 0,C 180,E1 -29897.803,E2 -29897.803} C_VEL
LIN {X 0,Y 75.072,Z 665.062,A -85,B 0,C 180,E1 -29891.303,E2 -29891.303} C_VEL
LIN {X 0,Y 92.051,Z 657.304,A -85,B 0,C 180,E1 -29887.011,E2 -29887.011} C_VEL
LIN {X 0,Y 107.485,Z 648.632,A -85,B 0,C 180,E1 -29884.363,E2 -29884.363} C_VEL
LIN {X 0,Y 121.352,Z 639.285,A -85,B 0,C 180,E1 -29882.553,E2 -29882.553} C_VEL
LIN {X 0,Y 133.566,Z 629.687,A -85,B 0,C 180,E1 -29881.327,E2 -29881.327} C_VEL
LIN {X 0,Y 145.833,Z 618.518,A -85,B 0,C 180,E1 -29880.404,E2 -29880.404} C_VEL
LIN {X 0,Y 156.064,Z 607.651,A -85,B 0,C 180,E1 -29879.666,E2 -29879.666} C_VEL
LIN {X 0,Y 159.066,Z 604.174,A -85,B 0,C 180,E1 -29879.447,E2 -29879.447} C_VEL
LIN {X 0,Y 147.632,Z 616.602,A -85,B 0,C 180,E1 -29878.577,E2 -29878.577} C_VEL
LIN {X 0,Y 135.419,Z 627.94,A -85,B 0,C 180,E1 -29877.472,E2 -29877.472} C_VEL
LIN {X 0,Y 123.278,Z 637.653,A -85,B 0,C 180,E1 -29876.075,E2 -29876.075} C_VEL
LIN {X 0,Y 109.488,Z 646.99,A -85,B 0,C 180,E1 -29874.228,E2 -29874.228} C_VEL
LIN {X 0,Y 95.838,Z 654.781,A -85,B 0,C 180,E1 -29871.864,E2 -29871.864} C_VEL
LIN {X 0,Y 82.412,Z 661.264,A -85,B 0,C 180,E1 -29868.723,E2 -29868.723} C_VEL
LIN {X 0,Y 69.299,Z 666.517,A -85,B 0,C 180,E1 -29864.459,E2 -29864.459} C_VEL
LIN {X 0,Y 55.985,Z 670.852,A -85,B 0,C 180,E1 -29857.876,E2 -29857.876} C_VEL
LIN {X 0,Y 42.306,Z 674.359,A -85,B 0,C 180,E1 -29846.16,E2 -29846.16} C_VEL
LIN {X 0,Y 33.049,Z 676.215,A -85,B 0,C 180,E1 -29829.639,E2 -29829.639} C_VEL
LIN {X 0,Y 27.786,Z 677.109,A -85,B 0,C 180,E1 -29804.65,E2 -29804.65} C_VEL
LIN {X 0,Y 27.237,Z 677.247,A -85,B 0,C 180,E1 -29789.999,E2 -29789.999} C_VEL
LIN {X 0,Y 29.775,Z 676.742,A -85,B 0,C 180,E1 -29761.83,E2 -29761.83} C_VEL
LIN {X 0,Y 37.317,Z 675.392,A -85,B 0,C 180,E1 -29741.12,E2 -29741.12} C_VEL
LIN {X 0,Y 47.838,Z 672.98,A -85,B 0,C 180,E1 -29728.179,E2 -29728.179} C_VEL
LIN {X 0,Y 59.814,Z 669.649,A -85,B 0,C 180,E1 -29719.951,E2 -29719.951} C_VEL
LIN {X 0,Y 75.817,Z 663.936,A -85,B 0,C 180,E1 -29713.268,E2 -29713.268} C_VEL
LIN {X 0,Y 92.466,Z 656.396,A -85,B 0,C 180,E1 -29708.855,E2 -29708.855} C_VEL
LIN {X 0,Y 107.787,Z 647.868,A -85,B 0,C 180,E1 -29706.104,E2 -29706.104} C_VEL
LIN {X 0,Y 121.559,Z 638.64,A -85,B 0,C 180,E1 -29704.201,E2 -29704.201} C_VEL
LIN {X 0,Y 132.432,Z 630.198,A -85,B 0,C 180,E1 -29702.914,E2 -29702.914} C_VEL
LIN {X 0,Y 144.144,Z 619.762,A -85,B 0,C 180,E1 -29701.792,E2 -29701.792} C_VEL
LIN {X 0,Y 154.636,Z 608.846,A -85,B 0,C 180,E1 -29700.943,E2 -29700.943} C_VEL
LIN {X 0,Y 159.593,Z 603.134,A -85,B 0,C 180,E1 -29700.578,E2 -29700.578} C_VEL
LIN {X 0,Y 152.64,Z 611.102,A -85,B 0,C 180,E1 -29700.127,E2 -29700.127} C_VEL
LIN {X 0,Y 152.122,Z 612.452,A -85,B 0,C 180,E1 -29700.096,E2 -29700.096} C_VEL
LIN {X 0,Y 152.122,Z 652.271,A -85,B 0,C 180,E1 -29700.096,E2 -29700.096} C_VEL
LIN {X 0,Y 121.475,Z 652.271,A -85,B 0,C 180,E1 -29699.799,E2 -29699.799} C_VEL
LIN {X 0,Y 119.476,Z 650.271,A -85,B 0,C 180,E1 -29699.774,E2 -29699.774} C_VEL
LIN {X 0,Y 119.476,Z 642.09,A -85,B 0,C 180,E1 -29699.774,E2 -29699.774} C_VEL
LIN {X 0,Y 119.484,Z 640.09,A -85,B 0,C 180,E1 -29700.705,E2 -29700.705} C_VEL
LIN {X 0,Y 119.493,Z 640.073,A -85,B 0,C 180,E1 -29700.99,E2 -29700.99} C_VEL
LIN {X 0,Y 105.521,Z 649.079,A -85,B 0,C 180,E1 -29702.514,E2 -29702.514} C_VEL
LIN {X 0,Y 91.635,Z 656.607,A -85,B 0,C 180,E1 -29704.412,E2 -29704.412} C_VEL
LIN {X 0,Y 77.904,Z 662.743,A -85,B 0,C 180,E1 -29707.091,E2 -29707.091} C_VEL
LIN {X 0,Y 64.396,Z 667.763,A -85,B 0,C 180,E1 -29710.815,E2 -29710.815} C_VEL
LIN {X 0,Y 51.255,Z 671.641,A -85,B 0,C 180,E1 -29716.295,E2 -29716.295} C_VEL
LIN {X 0,Y 38.803,Z 674.511,A -85,B 0,C 180,E1 -29725.096,E2 -29725.096} C_VEL
LIN {X 0,Y 27.935,Z 676.383,A -85,B 0,C 180,E1 -29740.996,E2 -29740.996} C_VEL
LIN {X 0,Y 20.979,Z 677.309,A -85,B 0,C 180,E1 -29770.427,E2 -29770.427} C_VEL
LIN {X 0,Y 20.131,Z 677.455,A -85,B 0,C 180,E1 -29789.999,E2 -29789.999} C_VEL
LIN {X 0,Y 23.724,Z 676.974,A -85,B 0,C 180,E1 -29826.331,E2 -29826.331} C_VEL
LIN {X 0,Y 33.033,Z 675.65,A -85,B 0,C 180,E1 -29848.323,E2 -29848.323} C_VEL
LIN {X 0,Y 44.886,Z 673.261,A -85,B 0,C 180,E1 -29859.955,E2 -29859.955} C_VEL
LIN {X 0,Y 57.756,Z 669.957,A -85,B 0,C 180,E1 -29866.769,E2 -29866.769} C_VEL
LIN {X 0,Y 74.491,Z 664.273,A -85,B 0,C 180,E1 -29872.15,E2 -29872.15} C_VEL
LIN {X 0,Y 91.632,Z 656.775,A -85,B 0,C 180,E1 -29875.611,E2 -29875.611} C_VEL
LIN {X 0,Y 107.257,Z 648.273,A -85,B 0,C 180,E1 -29877.775,E2 -29877.775} C_VEL
LIN {X 0,Y 119.49,Z 640.304,A -85,B 0,C 180,E1 -29879.077,E2 -29879.077} C_VEL
LIN {X 0,Y 119.483,Z 640.318,A -85,B 0,C 180,E1 -29879.31,E2 -29879.31} C_VEL
LIN {X 0,Y 105.427,Z 649.44,A -85,B 0,C 180,E1 -29880.719,E2 -29880.719} C_VEL
LIN {X 0,Y 91.452,Z 657.096,A -85,B 0,C 180,E1 -29882.535,E2 -29882.535} C_VEL
LIN {X 0,Y 76.342,Z 663.88,A -85,B 0,C 180,E1 -29885.281,E2 -29885.281} C_VEL
LIN {X 0,Y 60.598,Z 669.573,A -85,B 0,C 180,E1 -29889.667,E2 -29889.667} C_VEL
LIN {X 0,Y 50.679,Z 672.498,A -85,B 0,C 180,E1 -29893.897,E2 -29893.897} C_VEL
LIN {X 0,Y 38.119,Z 675.476,A -85,B 0,C 180,E1 -29902.803,E2 -29902.803} C_VEL
LIN {X 0,Y 27.144,Z 677.455,A -85,B 0,C 180,E1 -29919.038,E2 -29919.038} C_VEL
LIN {X 0,Y 20.408,Z 678.453,A -85,B 0,C 180,E1 -29949.857,E2 -29949.857} C_VEL
LIN {X 0,Y 19.878,Z 678.623,A -85,B 0,C 180,E1 -29970.001,E2 -29970.001} C_VEL
LIN {X 0,Y 22.992,Z 678.04,A -85,B 0,C 180,E1 -30007.687,E2 -30007.687} C_VEL
LIN {X 0,Y 32.343,Z 676.578,A -85,B 0,C 180,E1 -30030.365,E2 -30030.365} C_VEL
LIN {X 0,Y 44.275,Z 674.037,A -85,B 0,C 180,E1 -30042.253,E2 -30042.253} C_VEL
LIN {X 0,Y 60.602,Z 669.481,A -85,B 0,C 180,E1 -30050.313,E2 -30050.313} C_VEL
